Yaskawa INFORM job: A_ROOF_UPPER_0614_2_PAINT_12.JBI

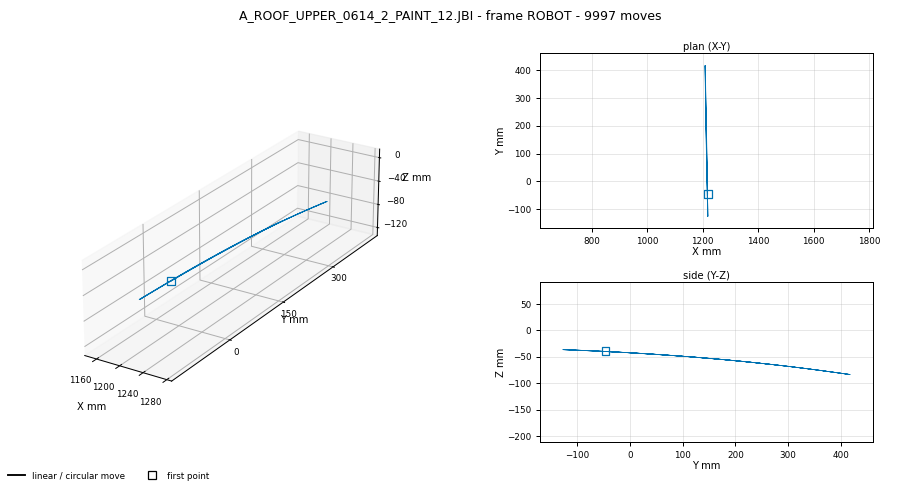
[picture p0: tool path of A_ROOF_UPPER_0614_2_PAINT_12.JBI in frame ROBOT, 9997 of 9997 moves have a stored position in this frame; points joined in program order, loops and branches not executed]
/JOB
//NAME A_ROOF_UPPER_0614_2_PAINT12
//POS
///NPOS 9997,0,0,0,0,0
///TOOL 1
///USER 0
///POSTYPE ROBOT
///RECTAN
///RCONF 1,0,0,0,0,0,0,0,0,0,0,0,0,0,0,0,0,0,0,0,0,0,0,0
C00000=1218.078,-45.969,-39.656,179.952,5.400,148.957
C00001=1218.073,-45.719,-39.668,179.954,5.400,148.956
C00002=1218.068,-45.469,-39.681,179.956,5.401,148.955
C00003=1218.063,-45.220,-39.693,179.959,5.401,148.955
C00004=1218.057,-44.970,-39.705,179.961,5.401,148.954
C00005=1218.052,-44.720,-39.718,179.964,5.401,148.953
C00006=1218.047,-44.471,-39.730,179.966,5.402,148.953
C00007=1218.042,-44.221,-39.742,179.968,5.401,148.952
C00008=1218.037,-43.971,-39.755,179.971,5.402,148.951
C00009=1218.032,-43.722,-39.768,179.973,5.401,148.950
C00010=1218.027,-43.472,-39.780,179.976,5.402,148.950
C00011=1218.022,-43.222,-39.792,179.979,5.402,148.949
C00012=1218.016,-42.973,-39.805,179.981,5.402,148.948
C00013=1218.012,-42.723,-39.818,179.983,5.403,148.948
C00014=1218.007,-42.474,-39.830,179.986,5.403,148.947
C00015=1218.001,-42.224,-39.842,179.988,5.403,148.946
C00016=1217.996,-41.974,-39.856,179.991,5.403,148.945
C00017=1217.990,-41.725,-39.868,179.993,5.404,148.945
C00018=1217.986,-41.475,-39.881,179.995,5.403,148.944
C00019=1217.980,-41.225,-39.893,179.998,5.404,148.943
C00020=1217.975,-40.976,-39.906,-180.000,5.403,148.943
C00021=1217.970,-40.726,-39.918,-179.997,5.404,148.942
C00022=1217.966,-40.476,-39.931,-179.995,5.405,148.942
C00023=1217.961,-40.227,-39.944,-179.993,5.404,148.941
C00024=1217.955,-39.977,-39.956,-179.990,5.405,148.940
C00025=1217.950,-39.728,-39.968,-179.988,5.405,148.939
C00026=1217.944,-39.478,-39.981,-179.985,5.405,148.939
C00027=1217.940,-39.228,-39.994,-179.983,5.406,148.938
C00028=1217.934,-38.979,-40.007,-179.980,5.406,148.937
C00029=1217.929,-38.729,-40.020,-179.978,5.406,148.937
C00030=1217.924,-38.480,-40.032,-179.975,5.406,148.936
C00031=1217.919,-38.229,-40.044,-179.973,5.407,148.935
C00032=1217.914,-37.980,-40.057,-179.971,5.406,148.935
C00033=1217.908,-37.731,-40.070,-179.968,5.407,148.934
C00034=1217.904,-37.481,-40.083,-179.965,5.407,148.933
C00035=1217.899,-37.231,-40.096,-179.963,5.407,148.932
C00036=1217.894,-36.982,-40.108,-179.961,5.407,148.932
C00037=1217.889,-36.733,-40.121,-179.959,5.407,148.931
C00038=1217.883,-36.482,-40.135,-179.956,5.408,148.930
C00039=1217.878,-36.233,-40.147,-179.953,5.408,148.930
C00040=1217.873,-35.984,-40.160,-179.951,5.408,148.929
C00041=1217.868,-35.734,-40.172,-179.948,5.408,148.928
C00042=1217.863,-35.484,-40.185,-179.946,5.409,148.928
C00043=1217.858,-35.235,-40.199,-179.944,5.408,148.927
C00044=1217.852,-34.985,-40.210,-179.941,5.409,148.926
C00045=1217.848,-34.735,-40.223,-179.938,5.409,148.925
C00046=1217.842,-34.485,-40.236,-179.937,5.409,148.925
C00047=1217.837,-34.236,-40.249,-179.934,5.410,148.924
C00048=1217.832,-33.986,-40.262,-179.931,5.410,148.924
C00049=1217.827,-33.736,-40.275,-179.929,5.410,148.923
C00050=1217.822,-33.487,-40.287,-179.927,5.411,148.922
C00051=1217.817,-33.237,-40.301,-179.924,5.411,148.921
C00052=1217.812,-32.988,-40.314,-179.922,5.411,148.921
C00053=1217.807,-32.739,-40.327,-179.919,5.411,148.920
C00054=1217.802,-32.489,-40.340,-179.917,5.412,148.919
C00055=1217.796,-32.239,-40.353,-179.915,5.411,148.919
C00056=1217.791,-31.990,-40.366,-179.912,5.412,148.918
C00057=1217.787,-31.740,-40.379,-179.909,5.412,148.917
C00058=1217.781,-31.490,-40.392,-179.907,5.412,148.917
C00059=1217.776,-31.241,-40.404,-179.904,5.412,148.916
C00060=1217.771,-30.991,-40.417,-179.902,5.413,148.915
C00061=1217.765,-30.741,-40.430,-179.900,5.413,148.914
C00062=1217.760,-30.492,-40.443,-179.897,5.413,148.914
C00063=1217.756,-30.242,-40.456,-179.894,5.414,148.913
C00064=1217.750,-29.992,-40.469,-179.892,5.413,148.912
C00065=1217.745,-29.743,-40.483,-179.890,5.414,148.912
C00066=1217.740,-29.493,-40.496,-179.887,5.414,148.911
C00067=1217.734,-29.244,-40.509,-179.885,5.414,148.910
C00068=1217.730,-28.994,-40.522,-179.882,5.414,148.910
C00069=1217.725,-28.745,-40.534,-179.880,5.415,148.909
C00070=1217.720,-28.494,-40.548,-179.878,5.415,148.908
C00071=1217.715,-28.246,-40.561,-179.875,5.415,148.908
C00072=1217.710,-27.996,-40.574,-179.873,5.416,148.907
C00073=1217.704,-27.746,-40.587,-179.870,5.416,148.906
C00074=1217.699,-27.497,-40.600,-179.868,5.416,148.906
C00075=1217.695,-27.247,-40.613,-179.865,5.417,148.905
C00076=1217.689,-26.998,-40.627,-179.863,5.417,148.904
C00077=1217.684,-26.748,-40.639,-179.861,5.417,148.904
C00078=1217.679,-26.498,-40.653,-179.858,5.417,148.903
C00079=1217.674,-26.249,-40.666,-179.855,5.418,148.902
C00080=1217.669,-25.999,-40.679,-179.853,5.417,148.901
C00081=1217.664,-25.750,-40.692,-179.851,5.418,148.901
C00082=1217.659,-25.499,-40.705,-179.848,5.418,148.900
C00083=1217.653,-25.250,-40.719,-179.846,5.418,148.899
C00084=1217.648,-25.001,-40.732,-179.843,5.419,148.899
C00085=1217.643,-24.751,-40.746,-179.840,5.419,148.898
C00086=1217.638,-24.502,-40.758,-179.838,5.420,148.897
C00087=1217.633,-24.251,-40.772,-179.836,5.419,148.897
C00088=1217.628,-24.002,-40.785,-179.833,5.420,148.896
C00089=1217.623,-23.752,-40.798,-179.830,5.420,148.895
C00090=1217.618,-23.503,-40.811,-179.828,5.420,148.894
C00091=1217.613,-23.253,-40.825,-179.826,5.420,148.894
C00092=1217.607,-22.984,-40.839,-179.823,5.421,148.893
C00093=1217.602,-22.715,-40.854,-179.820,5.421,148.892
C00094=1217.597,-22.445,-40.867,-179.818,5.421,148.892
C00095=1217.591,-22.176,-40.882,-179.816,5.422,148.891
C00096=1217.585,-21.926,-40.896,-179.813,5.422,148.890
C00097=1217.581,-21.677,-40.909,-179.810,5.423,148.890
C00098=1217.575,-21.427,-40.922,-179.808,5.422,148.889
C00099=1217.571,-21.177,-40.935,-179.806,5.423,148.888
C00100=1217.565,-20.928,-40.949,-179.803,5.423,148.888
C00101=1217.561,-20.678,-40.962,-179.800,5.424,148.887
C00102=1217.555,-20.429,-40.976,-179.798,5.423,148.886
C00103=1217.551,-20.179,-40.989,-179.795,5.424,148.885
C00104=1217.545,-19.929,-41.002,-179.793,5.424,148.885
C00105=1217.540,-19.680,-41.016,-179.791,5.424,148.884
C00106=1217.535,-19.430,-41.029,-179.788,5.425,148.883
C00107=1217.530,-19.180,-41.044,-179.785,5.425,148.883
C00108=1217.524,-18.931,-41.056,-179.783,5.426,148.882
C00109=1217.520,-18.681,-41.070,-179.781,5.425,148.881
C00110=1217.514,-18.432,-41.083,-179.778,5.426,148.881
C00111=1217.509,-18.182,-41.097,-179.775,5.426,148.880
C00112=1217.504,-17.933,-41.110,-179.773,5.426,148.879
C00113=1217.499,-17.683,-41.124,-179.771,5.427,148.879
C00114=1217.494,-17.434,-41.137,-179.768,5.427,148.878
C00115=1217.489,-17.184,-41.151,-179.766,5.428,148.877
C00116=1217.484,-16.934,-41.165,-179.764,5.427,148.877
C00117=1217.479,-16.685,-41.178,-179.761,5.428,148.876
C00118=1217.474,-16.435,-41.192,-179.758,5.428,148.875
C00119=1217.468,-16.186,-41.205,-179.756,5.428,148.875
C00120=1217.464,-15.936,-41.218,-179.754,5.429,148.874
C00121=1217.458,-15.687,-41.232,-179.751,5.429,148.873
C00122=1217.453,-15.437,-41.246,-179.748,5.430,148.872
C00123=1217.449,-15.187,-41.260,-179.746,5.429,148.872
C00124=1217.443,-14.938,-41.273,-179.744,5.430,148.871
C00125=1217.438,-14.688,-41.287,-179.741,5.430,148.870
C00126=1217.433,-14.439,-41.300,-179.738,5.431,148.870
C00127=1217.428,-14.189,-41.314,-179.736,5.431,148.869
C00128=1217.423,-13.939,-41.328,-179.734,5.431,148.868
C00129=1217.418,-13.690,-41.341,-179.731,5.432,148.868
C00130=1217.413,-13.440,-41.355,-179.729,5.431,148.867
C00131=1217.407,-13.191,-41.369,-179.726,5.432,148.866
C00132=1217.403,-12.941,-41.382,-179.724,5.432,148.866
C00133=1217.398,-12.691,-41.396,-179.721,5.433,148.865
C00134=1217.392,-12.442,-41.410,-179.719,5.433,148.864
C00135=1217.387,-12.192,-41.424,-179.717,5.433,148.864
C00136=1217.383,-11.943,-41.437,-179.714,5.434,148.863
C00137=1217.377,-11.694,-41.451,-179.711,5.434,148.862
C00138=1217.372,-11.443,-41.465,-179.709,5.434,148.862
C00139=1217.368,-11.194,-41.479,-179.707,5.434,148.861
C00140=1217.362,-10.945,-41.492,-179.704,5.435,148.860
C00141=1217.357,-10.695,-41.507,-179.701,5.435,148.860
C00142=1217.351,-10.446,-41.520,-179.699,5.435,148.859
C00143=1217.347,-10.196,-41.534,-179.697,5.436,148.858
C00144=1217.342,-9.946,-41.548,-179.694,5.436,148.857
C00145=1217.336,-9.697,-41.561,-179.691,5.437,148.857
C00146=1217.331,-9.447,-41.575,-179.689,5.436,148.856
C00147=1217.327,-9.198,-41.589,-179.686,5.437,148.855
C00148=1217.322,-8.948,-41.603,-179.684,5.437,148.855
C00149=1217.317,-8.699,-41.617,-179.681,5.438,148.854
C00150=1217.311,-8.449,-41.631,-179.679,5.438,148.853
C00151=1217.307,-8.199,-41.645,-179.676,5.438,148.853
C00152=1217.302,-7.950,-41.658,-179.674,5.439,148.852
C00153=1217.297,-7.701,-41.673,-179.672,5.439,148.851
C00154=1217.291,-7.450,-41.686,-179.670,5.439,148.851
C00155=1217.286,-7.201,-41.700,-179.667,5.440,148.850
C00156=1217.281,-6.951,-41.714,-179.664,5.440,148.849
C00157=1217.276,-6.702,-41.729,-179.662,5.441,148.849
C00158=1217.272,-6.452,-41.742,-179.660,5.440,148.848
C00159=1217.266,-6.203,-41.756,-179.657,5.441,148.847
C00160=1217.261,-5.954,-41.771,-179.654,5.441,148.847
C00161=1217.256,-5.703,-41.784,-179.652,5.442,148.846
C00162=1217.250,-5.454,-41.798,-179.649,5.442,148.845
C00163=1217.246,-5.205,-41.812,-179.647,5.442,148.845
C00164=1217.241,-4.955,-41.827,-179.644,5.443,148.844
C00165=1217.236,-4.705,-41.840,-179.641,5.443,148.843
C00166=1217.231,-4.456,-41.854,-179.639,5.444,148.842
C00167=1217.226,-4.207,-41.868,-179.637,5.443,148.842
C00168=1217.221,-3.957,-41.883,-179.634,5.444,148.841
C00169=1217.216,-3.707,-41.897,-179.632,5.445,148.841
C00170=1217.210,-3.458,-41.911,-179.629,5.445,148.840
C00171=1217.205,-3.208,-41.924,-179.627,5.445,148.839
C00172=1217.200,-2.958,-41.939,-179.625,5.445,148.839
C00173=1217.195,-2.709,-41.953,-179.622,5.446,148.838
C00174=1217.190,-2.460,-41.967,-179.619,5.446,148.837
C00175=1217.185,-2.210,-41.981,-179.617,5.446,148.837
C00176=1217.180,-1.960,-41.995,-179.615,5.447,148.836
C00177=1217.176,-1.711,-42.009,-179.612,5.447,148.835
C00178=1217.171,-1.461,-42.023,-179.609,5.448,148.834
C00179=1217.165,-1.212,-42.037,-179.607,5.448,148.834
C00180=1217.160,-0.962,-42.052,-179.604,5.448,148.833
C00181=1217.155,-0.713,-42.066,-179.602,5.448,148.832
C00182=1217.150,-0.463,-42.080,-179.599,5.449,148.832
C00183=1217.145,-0.213,-42.094,-179.597,5.449,148.831
C00184=1217.140,0.036,-42.108,-179.594,5.450,148.830
C00185=1217.135,0.286,-42.123,-179.592,5.450,148.830
C00186=1217.130,0.535,-42.138,-179.590,5.450,148.829
C00187=1217.125,0.784,-42.152,-179.587,5.451,148.828
C00188=1217.120,1.034,-42.166,-179.584,5.452,148.828
C00189=1217.115,1.283,-42.180,-179.582,5.451,148.827
C00190=1217.110,1.533,-42.194,-179.580,5.452,148.826
C00191=1217.105,1.782,-42.209,-179.577,5.452,148.826
C00192=1217.100,2.032,-42.223,-179.574,5.453,148.825
C00193=1217.095,2.282,-42.237,-179.572,5.453,148.824
C00194=1217.090,2.532,-42.251,-179.570,5.453,148.824
C00195=1217.084,2.781,-42.265,-179.567,5.453,148.823
C00196=1217.078,3.050,-42.282,-179.564,5.454,148.822
C00197=1217.073,3.319,-42.297,-179.562,5.455,148.822
C00198=1217.068,3.588,-42.312,-179.559,5.455,148.821
C00199=1217.063,3.857,-42.328,-179.556,5.456,148.820
C00200=1217.058,4.106,-42.342,-179.554,5.456,148.820
C00201=1217.053,4.356,-42.357,-179.551,5.457,148.819
C00202=1217.048,4.606,-42.371,-179.549,5.456,148.818
C00203=1217.043,4.854,-42.386,-179.546,5.457,148.817
C00204=1217.038,5.104,-42.400,-179.544,5.457,148.817
C00205=1217.032,5.354,-42.415,-179.541,5.458,148.816
C00206=1217.027,5.604,-42.429,-179.538,5.458,148.815
C00207=1217.022,5.853,-42.444,-179.536,5.458,148.815
C00208=1217.017,6.102,-42.458,-179.534,5.459,148.814
C00209=1217.012,6.352,-42.473,-179.531,5.459,148.813
C00210=1217.007,6.602,-42.487,-179.528,5.460,148.813
C00211=1217.002,6.852,-42.501,-179.526,5.460,148.812
C00212=1216.997,7.100,-42.516,-179.524,5.460,148.812
C00213=1216.992,7.350,-42.531,-179.521,5.461,148.811
C00214=1216.987,7.600,-42.545,-179.519,5.461,148.810
C00215=1216.982,7.849,-42.560,-179.516,5.462,148.809
C00216=1216.977,8.099,-42.574,-179.513,5.462,148.809
C00217=1216.972,8.348,-42.588,-179.511,5.463,148.808
C00218=1216.967,8.597,-42.603,-179.509,5.462,148.807
C00219=1216.962,8.847,-42.618,-179.506,5.463,148.807
C00220=1216.957,9.097,-42.633,-179.503,5.464,148.806
C00221=1216.952,9.346,-42.648,-179.501,5.464,148.805
C00222=1216.947,9.596,-42.662,-179.498,5.465,148.805
C00223=1216.942,9.846,-42.676,-179.496,5.464,148.804
C00224=1216.937,10.095,-42.692,-179.494,5.465,148.804
C00225=1216.932,10.345,-42.706,-179.491,5.466,148.803
C00226=1216.927,10.594,-42.720,-179.489,5.466,148.802
C00227=1216.922,10.843,-42.735,-179.486,5.467,148.801
C00228=1216.917,11.093,-42.750,-179.483,5.467,148.801
C00229=1216.912,11.343,-42.765,-179.481,5.467,148.800
C00230=1216.907,11.592,-42.779,-179.479,5.467,148.799
C00231=1216.901,11.841,-42.793,-179.476,5.468,148.799
C00232=1216.897,12.090,-42.808,-179.473,5.469,148.798
C00233=1216.891,12.340,-42.823,-179.471,5.469,148.797
C00234=1216.886,12.590,-42.838,-179.468,5.470,148.797
C00235=1216.881,12.839,-42.852,-179.466,5.469,148.796
C00236=1216.876,13.089,-42.868,-179.464,5.470,148.796
C00237=1216.871,13.338,-42.882,-179.461,5.471,148.795
C00238=1216.866,13.588,-42.897,-179.458,5.471,148.794
C00239=1216.861,13.837,-42.912,-179.456,5.472,148.793
C00240=1216.856,14.087,-42.926,-179.453,5.472,148.793
C00241=1216.851,14.336,-42.941,-179.450,5.473,148.792
C00242=1216.847,14.587,-42.956,-179.448,5.472,148.791
C00243=1216.841,14.836,-42.972,-179.446,5.473,148.791
C00244=1216.836,15.086,-42.986,-179.443,5.474,148.790
C00245=1216.832,15.335,-43.001,-179.440,5.474,148.789
C00246=1216.826,15.584,-43.017,-179.438,5.475,148.789
C00247=1216.821,15.834,-43.031,-179.436,5.475,148.788
C00248=1216.817,16.083,-43.046,-179.434,5.475,148.788
C00249=1216.811,16.333,-43.061,-179.431,5.476,148.787
C00250=1216.806,16.582,-43.076,-179.428,5.476,148.786
C00251=1216.802,16.832,-43.090,-179.426,5.477,148.785
C00252=1216.796,17.081,-43.106,-179.423,5.477,148.785
C00253=1216.791,17.330,-43.121,-179.420,5.478,148.784
C00254=1216.787,17.580,-43.135,-179.418,5.478,148.783
C00255=1216.781,17.830,-43.150,-179.416,5.478,148.783
C00256=1216.776,18.079,-43.165,-179.413,5.479,148.782
C00257=1216.771,18.329,-43.180,-179.411,5.479,148.782
C00258=1216.766,18.578,-43.195,-179.408,5.480,148.781
C00259=1216.761,18.827,-43.210,-179.406,5.481,148.780
C00260=1216.756,19.078,-43.225,-179.403,5.481,148.780
C00261=1216.752,19.327,-43.240,-179.400,5.482,148.779
C00262=1216.746,19.577,-43.255,-179.398,5.481,148.778
C00263=1216.741,19.826,-43.270,-179.396,5.482,148.778
C00264=1216.736,20.075,-43.286,-179.393,5.482,148.777
C00265=1216.731,20.325,-43.300,-179.390,5.483,148.776
C00266=1216.726,20.574,-43.315,-179.388,5.483,148.775
C00267=1216.721,20.823,-43.331,-179.385,5.484,148.775
C00268=1216.716,21.073,-43.345,-179.383,5.485,148.774
C00269=1216.711,21.322,-43.361,-179.380,5.485,148.774
C00270=1216.707,21.572,-43.376,-179.378,5.485,148.773
C00271=1216.701,21.822,-43.392,-179.375,5.486,148.772
C00272=1216.696,22.071,-43.406,-179.373,5.486,148.772
C00273=1216.691,22.321,-43.421,-179.370,5.487,148.771
C00274=1216.686,22.570,-43.436,-179.367,5.487,148.770
C00275=1216.681,22.819,-43.452,-179.365,5.488,148.770
C00276=1216.676,23.069,-43.466,-179.363,5.489,148.769
C00277=1216.671,23.319,-43.482,-179.360,5.489,148.768
C00278=1216.666,23.568,-43.497,-179.357,5.490,148.768
C00279=1216.661,23.818,-43.513,-179.355,5.489,148.767
C00280=1216.656,24.067,-43.528,-179.353,5.490,148.766
C00281=1216.651,24.317,-43.543,-179.350,5.490,148.766
C00282=1216.646,24.566,-43.558,-179.347,5.491,148.765
C00283=1216.641,24.816,-43.574,-179.345,5.492,148.764
C00284=1216.637,25.065,-43.589,-179.342,5.492,148.764
C00285=1216.631,25.314,-43.604,-179.340,5.493,148.763
C00286=1216.626,25.564,-43.620,-179.337,5.494,148.763
C00287=1216.621,25.813,-43.635,-179.335,5.494,148.762
C00288=1216.616,26.064,-43.650,-179.333,5.494,148.761
C00289=1216.612,26.313,-43.665,-179.330,5.494,148.761
C00290=1216.606,26.562,-43.681,-179.327,5.495,148.760
C00291=1216.601,26.811,-43.696,-179.325,5.495,148.759
C00292=1216.596,27.061,-43.711,-179.322,5.496,148.758
C00293=1216.591,27.311,-43.727,-179.319,5.496,148.758
C00294=1216.587,27.560,-43.742,-179.317,5.497,148.757
C00295=1216.581,27.809,-43.758,-179.315,5.498,148.757
C00296=1216.576,28.059,-43.773,-179.312,5.498,148.756
C00297=1216.571,28.308,-43.788,-179.309,5.499,148.755
C00298=1216.566,28.558,-43.804,-179.307,5.499,148.755
C00299=1216.562,28.807,-43.819,-179.305,5.499,148.754
C00300=1216.556,29.076,-43.836,-179.302,5.500,148.753
C00301=1216.550,29.344,-43.853,-179.299,5.500,148.753
C00302=1216.545,29.613,-43.870,-179.297,5.501,148.752
C00303=1216.540,29.882,-43.885,-179.293,5.502,148.751
C00304=1216.535,30.132,-43.901,-179.291,5.502,148.751
C00305=1216.530,30.381,-43.917,-179.289,5.502,148.750
C00306=1216.525,30.630,-43.932,-179.286,5.503,148.749
C00307=1216.519,30.880,-43.947,-179.283,5.503,148.749
C00308=1216.515,31.130,-43.963,-179.281,5.504,148.748
C00309=1216.510,31.378,-43.979,-179.279,5.505,148.747
C00310=1216.505,31.628,-43.995,-179.276,5.505,148.747
C00311=1216.500,31.877,-44.010,-179.273,5.506,148.746
C00312=1216.496,32.127,-44.026,-179.271,5.507,148.745
C00313=1216.490,32.376,-44.041,-179.268,5.507,148.745
C00314=1216.485,32.626,-44.057,-179.265,5.508,148.744
C00315=1216.480,32.876,-44.073,-179.263,5.508,148.743
C00316=1216.475,33.125,-44.088,-179.261,5.508,148.743
C00317=1216.470,33.374,-44.103,-179.259,5.509,148.742
C00318=1216.465,33.624,-44.119,-179.256,5.509,148.742
C00319=1216.460,33.873,-44.136,-179.253,5.510,148.741
C00320=1216.455,34.122,-44.151,-179.251,5.510,148.740
C00321=1216.450,34.372,-44.166,-179.248,5.511,148.740
C00322=1216.445,34.622,-44.182,-179.245,5.511,148.739
C00323=1216.440,34.871,-44.198,-179.243,5.512,148.738
C00324=1216.435,35.120,-44.213,-179.241,5.513,148.738
C00325=1216.431,35.370,-44.229,-179.238,5.513,148.737
C00326=1216.425,35.619,-44.245,-179.235,5.514,148.736
C00327=1216.420,35.869,-44.261,-179.233,5.515,148.736
C00328=1216.415,36.119,-44.277,-179.230,5.515,148.735
C00329=1216.411,36.368,-44.292,-179.227,5.516,148.734
C00330=1216.406,36.617,-44.308,-179.225,5.517,148.734
C00331=1216.401,36.867,-44.324,-179.223,5.517,148.733
C00332=1216.395,37.116,-44.339,-179.220,5.517,148.733
C00333=1216.390,37.366,-44.355,-179.218,5.517,148.732
C00334=1216.385,37.615,-44.372,-179.215,5.518,148.731
C00335=1216.381,37.864,-44.387,-179.213,5.518,148.731
C00336=1216.376,38.114,-44.403,-179.210,5.519,148.730
C00337=1216.371,38.364,-44.418,-179.208,5.520,148.729
C00338=1216.366,38.612,-44.434,-179.205,5.520,148.729
C00339=1216.361,38.862,-44.450,-179.202,5.521,148.728
C00340=1216.355,39.112,-44.466,-179.200,5.522,148.727
C00341=1216.351,39.361,-44.483,-179.197,5.522,148.727
C00342=1216.345,39.611,-44.498,-179.195,5.523,148.726
C00343=1216.341,39.860,-44.513,-179.192,5.523,148.725
C00344=1216.336,40.109,-44.530,-179.190,5.524,148.725
C00345=1216.331,40.359,-44.545,-179.187,5.525,148.724
C00346=1216.326,40.609,-44.561,-179.184,5.525,148.724
C00347=1216.321,40.858,-44.578,-179.182,5.526,148.723
C00348=1216.316,41.107,-44.593,-179.179,5.526,148.722
C00349=1216.311,41.357,-44.609,-179.177,5.527,148.722
C00350=1216.306,41.606,-44.626,-179.174,5.528,148.721
C00351=1216.301,41.856,-44.642,-179.172,5.528,148.720
C00352=1216.296,42.105,-44.658,-179.169,5.529,148.720
C00353=1216.291,42.355,-44.674,-179.166,5.529,148.719
C00354=1216.286,42.604,-44.689,-179.164,5.530,148.718
C00355=1216.281,42.853,-44.706,-179.161,5.530,148.718
C00356=1216.276,43.103,-44.722,-179.159,5.531,148.717
C00357=1216.271,43.352,-44.738,-179.157,5.531,148.717
C00358=1216.266,43.602,-44.754,-179.154,5.532,148.716
C00359=1216.261,43.851,-44.770,-179.152,5.532,148.715
C00360=1216.256,44.101,-44.786,-179.149,5.533,148.715
C00361=1216.251,44.350,-44.802,-179.146,5.533,148.714
C00362=1216.246,44.600,-44.818,-179.144,5.534,148.713
C00363=1216.241,44.849,-44.835,-179.142,5.535,148.713
C00364=1216.236,45.099,-44.851,-179.139,5.535,148.712
C00365=1216.231,45.347,-44.867,-179.136,5.536,148.711
C00366=1216.227,45.598,-44.883,-179.134,5.536,148.711
C00367=1216.222,45.846,-44.899,-179.131,5.537,148.710
C00368=1216.217,46.096,-44.915,-179.129,5.538,148.710
C00369=1216.212,46.345,-44.931,-179.126,5.538,148.709
C00370=1216.207,46.595,-44.947,-179.124,5.539,148.708
C00371=1216.202,46.844,-44.964,-179.121,5.540,148.708
C00372=1216.197,47.094,-44.980,-179.118,5.540,148.707
C00373=1216.192,47.343,-44.996,-179.116,5.541,148.707
C00374=1216.187,47.592,-45.013,-179.114,5.542,148.706
C00375=1216.182,47.842,-45.028,-179.111,5.542,148.705
C00376=1216.178,48.091,-45.045,-179.108,5.543,148.705
C00377=1216.172,48.340,-45.061,-179.106,5.543,148.704
C00378=1216.168,48.590,-45.077,-179.103,5.544,148.703
C00379=1216.162,48.839,-45.094,-179.101,5.545,148.703
C00380=1216.157,49.089,-45.111,-179.098,5.545,148.702
C00381=1216.152,49.338,-45.126,-179.096,5.546,148.701
C00382=1216.148,49.588,-45.143,-179.093,5.546,148.701
C00383=1216.143,49.838,-45.159,-179.090,5.547,148.700
C00384=1216.138,50.087,-45.175,-179.088,5.548,148.700
C00385=1216.133,50.336,-45.192,-179.086,5.548,148.699
C00386=1216.128,50.585,-45.208,-179.083,5.549,148.698
C00387=1216.123,50.835,-45.225,-179.080,5.549,148.698
C00388=1216.118,51.084,-45.241,-179.078,5.550,148.697
C00389=1216.113,51.334,-45.258,-179.075,5.551,148.696
C00390=1216.108,51.584,-45.274,-179.073,5.551,148.696
C00391=1216.103,51.832,-45.290,-179.070,5.552,148.695
C00392=1216.099,52.082,-45.307,-179.068,5.553,148.695
C00393=1216.093,52.331,-45.324,-179.065,5.553,148.694
C00394=1216.088,52.581,-45.340,-179.062,5.554,148.693
C00395=1216.084,52.831,-45.356,-179.060,5.555,148.693
C00396=1216.079,53.079,-45.373,-179.058,5.555,148.692
C00397=1216.074,53.329,-45.389,-179.055,5.556,148.691
C00398=1216.068,53.578,-45.406,-179.052,5.556,148.691
C00399=1216.063,53.828,-45.422,-179.050,5.557,148.690
C00400=1216.059,54.078,-45.439,-179.047,5.559,148.690
C00401=1216.054,54.326,-45.455,-179.044,5.559,148.689
C00402=1216.049,54.576,-45.472,-179.042,5.560,148.688
C00403=1216.044,54.826,-45.489,-179.039,5.560,148.688
C00404=1216.039,55.094,-45.506,-179.036,5.561,148.687
C00405=1216.033,55.362,-45.524,-179.034,5.561,148.686
C00406=1216.028,55.631,-45.542,-179.031,5.562,148.686
C00407=1216.022,55.899,-45.559,-179.028,5.562,148.685
C00408=1216.018,56.149,-45.576,-179.026,5.563,148.684
C00409=1216.013,56.399,-45.593,-179.024,5.564,148.684
C00410=1216.008,56.647,-45.610,-179.021,5.564,148.683
C00411=1216.003,56.897,-45.626,-179.018,5.566,148.683
C00412=1215.998,57.147,-45.644,-179.015,5.566,148.682
C00413=1215.993,57.395,-45.660,-179.013,5.567,148.681
C00414=1215.988,57.645,-45.677,-179.010,5.568,148.681
C00415=1215.983,57.895,-45.694,-179.008,5.568,148.680
C00416=1215.978,58.143,-45.710,-179.005,5.569,148.679
C00417=1215.974,58.393,-45.727,-179.003,5.570,148.679
C00418=1215.968,58.643,-45.744,-179.000,5.571,148.678
C00419=1215.963,58.892,-45.760,-178.998,5.571,148.678
C00420=1215.959,59.141,-45.777,-178.995,5.572,148.677
C00421=1215.954,59.391,-45.794,-178.992,5.572,148.676
C00422=1215.949,59.640,-45.811,-178.990,5.573,148.676
C00423=1215.944,59.889,-45.827,-178.988,5.574,148.675
C00424=1215.939,60.139,-45.845,-178.985,5.574,148.675
C00425=1215.934,60.388,-45.861,-178.982,5.575,148.674
C00426=1215.929,60.637,-45.878,-178.980,5.575,148.673
C00427=1215.924,60.887,-45.895,-178.978,5.576,148.673
C00428=1215.920,61.136,-45.911,-178.975,5.577,148.672
C00429=1215.914,61.386,-45.929,-178.972,5.577,148.671
C00430=1215.909,61.635,-45.945,-178.969,5.579,148.671
C00431=1215.904,61.885,-45.962,-178.967,5.579,148.670
C00432=1215.900,62.134,-45.979,-178.964,5.580,148.670
C00433=1215.895,62.384,-45.996,-178.962,5.581,148.669
C00434=1215.889,62.633,-46.013,-178.959,5.581,148.668
C00435=1215.885,62.882,-46.030,-178.957,5.582,148.668
C00436=1215.880,63.132,-46.047,-178.954,5.583,148.667
C00437=1215.875,63.381,-46.064,-178.952,5.583,148.667
C00438=1215.870,63.630,-46.081,-178.949,5.584,148.666
C00439=1215.865,63.880,-46.097,-178.946,5.585,148.665
C00440=1215.860,64.129,-46.115,-178.944,5.586,148.665
C00441=1215.855,64.379,-46.131,-178.942,5.586,148.664
C00442=1215.850,64.627,-46.149,-178.939,5.587,148.664
C00443=1215.845,64.877,-46.166,-178.936,5.587,148.663
C00444=1215.840,65.127,-46.183,-178.934,5.589,148.662
C00445=1215.836,65.376,-46.200,-178.931,5.590,148.662
C00446=1215.830,65.626,-46.217,-178.928,5.590,148.661
C00447=1215.826,65.874,-46.234,-178.926,5.591,148.660
C00448=1215.820,66.124,-46.251,-178.924,5.592,148.660
C00449=1215.816,66.373,-46.268,-178.921,5.592,148.659
C00450=1215.811,66.623,-46.285,-178.918,5.593,148.659
C00451=1215.807,66.872,-46.302,-178.916,5.593,148.658
C00452=1215.801,67.122,-46.320,-178.914,5.594,148.658
C00453=1215.796,67.371,-46.336,-178.911,5.595,148.657
C00454=1215.791,67.620,-46.353,-178.908,5.595,148.656
C00455=1215.787,67.869,-46.371,-178.905,5.597,148.656
C00456=1215.782,68.119,-46.388,-178.903,5.598,148.655
C00457=1215.777,68.369,-46.405,-178.900,5.598,148.655
C00458=1215.772,68.618,-46.423,-178.898,5.599,148.654
C00459=1215.767,68.867,-46.439,-178.895,5.599,148.653
C00460=1215.762,69.116,-46.456,-178.893,5.600,148.653
C00461=1215.757,69.365,-46.474,-178.890,5.601,148.652
C00462=1215.753,69.615,-46.491,-178.888,5.601,148.651
C00463=1215.747,69.865,-46.508,-178.885,5.602,148.651
C00464=1215.743,70.114,-46.526,-178.883,5.603,148.650
C00465=1215.738,70.363,-46.543,-178.880,5.604,148.650
C00466=1215.733,70.613,-46.561,-178.877,5.605,148.649
C00467=1215.728,70.861,-46.577,-178.875,5.605,148.648
C00468=1215.723,71.111,-46.594,-178.872,5.606,148.648
C00469=1215.718,71.360,-46.612,-178.870,5.607,148.647
C00470=1215.713,71.610,-46.629,-178.867,5.608,148.647
C00471=1215.709,71.859,-46.647,-178.865,5.608,148.646
C00472=1215.703,72.109,-46.664,-178.862,5.609,148.646
C00473=1215.699,72.358,-46.681,-178.860,5.610,148.645
C00474=1215.694,72.607,-46.699,-178.857,5.611,148.644
C00475=1215.689,72.857,-46.716,-178.854,5.612,148.644
C00476=1215.684,73.106,-46.734,-178.852,5.612,148.643
C00477=1215.679,73.355,-46.750,-178.849,5.613,148.642
C00478=1215.674,73.604,-46.768,-178.847,5.614,148.642
C00479=1215.669,73.854,-46.786,-178.844,5.615,148.641
C00480=1215.664,74.103,-46.803,-178.842,5.615,148.641
C00481=1215.659,74.353,-46.820,-178.839,5.616,148.640
C00482=1215.654,74.602,-46.838,-178.836,5.617,148.640
C00483=1215.649,74.851,-46.856,-178.834,5.618,148.639
C00484=1215.645,75.101,-46.873,-178.831,5.619,148.638
C00485=1215.640,75.350,-46.891,-178.829,5.619,148.638
C00486=1215.635,75.600,-46.908,-178.826,5.620,148.637
C00487=1215.631,75.849,-46.925,-178.824,5.621,148.637
C00488=1215.625,76.098,-46.943,-178.821,5.621,148.636
C00489=1215.620,76.347,-46.961,-178.818,5.623,148.636
C00490=1215.616,76.597,-46.979,-178.816,5.624,148.635
C00491=1215.610,76.846,-46.996,-178.813,5.624,148.634
C00492=1215.606,77.095,-47.013,-178.811,5.625,148.634
C00493=1215.601,77.345,-47.031,-178.808,5.626,148.633
C00494=1215.596,77.594,-47.049,-178.806,5.626,148.632
C00495=1215.591,77.843,-47.067,-178.803,5.627,148.632
C00496=1215.586,78.093,-47.084,-178.800,5.629,148.631
C00497=1215.582,78.342,-47.101,-178.798,5.629,148.631
C00498=1215.577,78.591,-47.119,-178.795,5.630,148.630
C00499=1215.572,78.841,-47.136,-178.793,5.630,148.629
C00500=1215.567,79.090,-47.154,-178.790,5.631,148.629
C00501=1215.562,79.339,-47.172,-178.788,5.632,148.628
C00502=1215.557,79.589,-47.190,-178.785,5.633,148.628
C00503=1215.552,79.838,-47.207,-178.783,5.634,148.627
C00504=1215.547,80.087,-47.225,-178.780,5.635,148.627
C00505=1215.543,80.336,-47.243,-178.777,5.635,148.626
C00506=1215.537,80.586,-47.260,-178.775,5.636,148.626
C00507=1215.532,80.835,-47.278,-178.772,5.637,148.625
C00508=1215.527,81.104,-47.298,-178.769,5.638,148.624
C00509=1215.522,81.373,-47.316,-178.767,5.639,148.624
C00510=1215.517,81.641,-47.336,-178.764,5.639,148.623
C00511=1215.512,81.909,-47.355,-178.761,5.641,148.622
C00512=1215.507,82.158,-47.373,-178.759,5.642,148.622
C00513=1215.502,82.408,-47.390,-178.756,5.642,148.621
C00514=1215.497,82.657,-47.408,-178.753,5.643,148.621
C00515=1215.492,82.906,-47.426,-178.751,5.644,148.620
C00516=1215.487,83.156,-47.444,-178.748,5.645,148.619
C00517=1215.482,83.405,-47.462,-178.746,5.646,148.619
C00518=1215.477,83.654,-47.480,-178.743,5.647,148.618
C00519=1215.473,83.903,-47.497,-178.741,5.647,148.618
C00520=1215.468,84.153,-47.515,-178.738,5.648,148.617
C00521=1215.463,84.402,-47.533,-178.736,5.648,148.616
C00522=1215.458,84.651,-47.551,-178.733,5.650,148.616
C00523=1215.454,84.901,-47.569,-178.730,5.651,148.615
C00524=1215.449,85.150,-47.587,-178.728,5.651,148.615
C00525=1215.444,85.399,-47.605,-178.725,5.652,148.614
C00526=1215.439,85.648,-47.623,-178.723,5.653,148.614
C00527=1215.434,85.897,-47.641,-178.720,5.654,148.613
C00528=1215.429,86.147,-47.659,-178.717,5.655,148.613
C00529=1215.424,86.396,-47.677,-178.715,5.656,148.612
C00530=1215.419,86.645,-47.695,-178.712,5.656,148.611
C00531=1215.415,86.895,-47.713,-178.710,5.657,148.611
C00532=1215.410,87.144,-47.731,-178.707,5.659,148.610
C00533=1215.405,87.394,-47.749,-178.704,5.659,148.609
C00534=1215.399,87.643,-47.767,-178.702,5.660,148.609
C00535=1215.394,87.893,-47.785,-178.700,5.661,148.608
C00536=1215.390,88.141,-47.804,-178.697,5.661,148.608
C00537=1215.385,88.391,-47.822,-178.694,5.663,148.607
C00538=1215.380,88.640,-47.840,-178.692,5.664,148.607
C00539=1215.375,88.889,-47.858,-178.689,5.664,148.606
C00540=1215.370,89.138,-47.876,-178.687,5.665,148.606
C00541=1215.366,89.388,-47.894,-178.684,5.666,148.605
C00542=1215.361,89.637,-47.912,-178.682,5.668,148.605
C00543=1215.356,89.887,-47.931,-178.679,5.668,148.604
C00544=1215.351,90.136,-47.949,-178.676,5.669,148.603
C00545=1215.346,90.385,-47.967,-178.674,5.670,148.603
C00546=1215.341,90.635,-47.985,-178.672,5.670,148.602
C00547=1215.336,90.884,-48.003,-178.668,5.672,148.602
C00548=1215.332,91.134,-48.021,-178.666,5.673,148.601
C00549=1215.327,91.382,-48.040,-178.664,5.673,148.600
C00550=1215.322,91.631,-48.058,-178.661,5.674,148.600
C00551=1215.317,91.881,-48.076,-178.658,5.676,148.599
C00552=1215.312,92.130,-48.095,-178.656,5.676,148.599
C00553=1215.307,92.380,-48.113,-178.653,5.677,148.598
C00554=1215.302,92.629,-48.131,-178.651,5.678,148.598
C00555=1215.298,92.878,-48.150,-178.648,5.678,148.597
C00556=1215.293,93.127,-48.168,-178.645,5.680,148.596
C00557=1215.289,93.377,-48.186,-178.643,5.681,148.596
C00558=1215.283,93.626,-48.205,-178.640,5.681,148.595
C00559=1215.278,93.875,-48.223,-178.638,5.682,148.595
C00560=1215.273,94.124,-48.241,-178.635,5.684,148.594
C00561=1215.269,94.374,-48.260,-178.632,5.684,148.594
C00562=1215.264,94.623,-48.278,-178.630,5.685,148.593
C00563=1215.258,94.872,-48.296,-178.628,5.686,148.593
C00564=1215.254,95.121,-48.315,-178.624,5.687,148.592
C00565=1215.250,95.371,-48.333,-178.622,5.688,148.591
C00566=1215.245,95.620,-48.351,-178.620,5.689,148.591
C00567=1215.239,95.870,-48.370,-178.618,5.690,148.590
C00568=1215.235,96.119,-48.389,-178.614,5.691,148.590
C00569=1215.230,96.368,-48.407,-178.612,5.692,148.589
C00570=1215.224,96.617,-48.425,-178.610,5.693,148.589
C00571=1215.220,96.866,-48.444,-178.607,5.693,148.588
C00572=1215.216,97.116,-48.462,-178.604,5.695,148.587
C00573=1215.211,97.365,-48.480,-178.602,5.696,148.587
C00574=1215.205,97.614,-48.500,-178.599,5.696,148.586
C00575=1215.201,97.864,-48.518,-178.597,5.697,148.586
C00576=1215.196,98.112,-48.537,-178.594,5.699,148.585
C00577=1215.191,98.362,-48.555,-178.591,5.699,148.585
C00578=1215.186,98.612,-48.574,-178.589,5.700,148.584
C00579=1215.182,98.860,-48.592,-178.586,5.701,148.584
C00580=1215.176,99.110,-48.611,-178.584,5.702,148.583
C00581=1215.172,99.359,-48.630,-178.581,5.703,148.583
C00582=1215.167,99.608,-48.648,-178.578,5.704,148.582
C00583=1215.162,99.858,-48.667,-178.576,5.705,148.581
C00584=1215.158,100.107,-48.686,-178.573,5.706,148.581
C00585=1215.153,100.356,-48.704,-178.571,5.707,148.580
C00586=1215.147,100.605,-48.723,-178.568,5.708,148.580
C00587=1215.143,100.855,-48.741,-178.565,5.709,148.579
C00588=1215.138,101.104,-48.760,-178.563,5.710,148.579
C00589=1215.133,101.354,-48.779,-178.560,5.710,148.578
C00590=1215.129,101.602,-48.798,-178.558,5.711,148.578
C00591=1215.123,101.852,-48.816,-178.555,5.713,148.577
C00592=1215.119,102.101,-48.835,-178.553,5.713,148.576
C00593=1215.113,102.350,-48.854,-178.550,5.714,148.576
C00594=1215.109,102.599,-48.872,-178.547,5.716,148.575
C00595=1215.104,102.849,-48.891,-178.545,5.717,148.575
C00596=1215.099,103.098,-48.910,-178.542,5.717,148.574
C00597=1215.095,103.347,-48.929,-178.540,5.718,148.574
C00598=1215.090,103.596,-48.948,-178.537,5.720,148.573
C00599=1215.085,103.845,-48.966,-178.535,5.720,148.573
C00600=1215.080,104.095,-48.985,-178.532,5.721,148.572
C00601=1215.075,104.344,-49.004,-178.529,5.723,148.572
C00602=1215.071,104.593,-49.024,-178.527,5.724,148.571
C00603=1215.066,104.842,-49.042,-178.525,5.724,148.570
C00604=1215.061,105.092,-49.061,-178.522,5.725,148.570
C00605=1215.056,105.341,-49.080,-178.519,5.727,148.569
C00606=1215.051,105.590,-49.099,-178.517,5.727,148.569
C00607=1215.047,105.839,-49.118,-178.514,5.728,148.568
C00608=1215.041,106.088,-49.137,-178.511,5.730,148.568
C00609=1215.037,106.338,-49.155,-178.509,5.730,148.567
C00610=1215.032,106.587,-49.175,-178.507,5.731,148.567
C00611=1215.028,106.836,-49.194,-178.503,5.733,148.566
C00612=1215.022,107.105,-49.214,-178.501,5.734,148.566
C00613=1215.017,107.373,-49.235,-178.498,5.735,148.565
C00614=1215.011,107.642,-49.255,-178.495,5.736,148.564
C00615=1215.007,107.910,-49.275,-178.492,5.737,148.564
C00616=1215.002,108.159,-49.295,-178.490,5.738,148.563
C00617=1214.997,108.409,-49.314,-178.488,5.739,148.563
C00618=1214.992,108.658,-49.332,-178.485,5.740,148.562
C00619=1214.987,108.908,-49.352,-178.482,5.741,148.562
C00620=1214.983,109.156,-49.371,-178.480,5.741,148.561
C00621=1214.978,109.406,-49.390,-178.477,5.743,148.561
C00622=1214.972,109.655,-49.409,-178.474,5.744,148.560
C00623=1214.968,109.904,-49.428,-178.472,5.745,148.559
C00624=1214.963,110.153,-49.447,-178.469,5.746,148.559
C00625=1214.959,110.402,-49.466,-178.467,5.747,148.558
C00626=1214.953,110.651,-49.485,-178.464,5.748,148.558
C00627=1214.949,110.901,-49.505,-178.462,5.750,148.557
C00628=1214.944,111.149,-49.524,-178.459,5.750,148.557
C00629=1214.939,111.400,-49.543,-178.457,5.751,148.556
C00630=1214.934,111.649,-49.562,-178.454,5.753,148.556
C00631=1214.930,111.898,-49.581,-178.451,5.753,148.555
C00632=1214.924,112.147,-49.600,-178.449,5.754,148.555
C00633=1214.920,112.396,-49.620,-178.446,5.756,148.554
C00634=1214.916,112.645,-49.639,-178.444,5.756,148.554
C00635=1214.910,112.894,-49.658,-178.441,5.757,148.553
C00636=1214.905,113.144,-49.678,-178.438,5.759,148.553
C00637=1214.901,113.392,-49.697,-178.436,5.759,148.552
C00638=1214.896,113.642,-49.716,-178.434,5.760,148.552
C00639=1214.891,113.891,-49.736,-178.430,5.762,148.551
C00640=1214.886,114.140,-49.755,-178.428,5.763,148.550
C00641=1214.882,114.390,-49.774,-178.426,5.763,148.550
C00642=1214.877,114.639,-49.794,-178.423,5.765,148.549
C00643=1214.872,114.888,-49.813,-178.420,5.766,148.549
C00644=1214.867,115.137,-49.833,-178.418,5.766,148.548
C00645=1214.863,115.386,-49.852,-178.415,5.768,148.548
C00646=1214.858,115.636,-49.871,-178.412,5.769,148.547
C00647=1214.853,115.885,-49.891,-178.410,5.770,148.547
C00648=1214.848,116.134,-49.910,-178.407,5.771,148.546
C00649=1214.842,116.383,-49.930,-178.405,5.772,148.546
C00650=1214.838,116.632,-49.949,-178.402,5.774,148.545
C00651=1214.834,116.882,-49.968,-178.400,5.775,148.545
C00652=1214.828,117.131,-49.988,-178.397,5.775,148.544
C00653=1214.824,117.380,-50.007,-178.394,5.777,148.544
C00654=1214.818,117.629,-50.027,-178.392,5.778,148.543
C00655=1214.814,117.879,-50.046,-178.390,5.778,148.543
C00656=1214.810,118.128,-50.065,-178.387,5.780,148.542
C00657=1214.804,118.376,-50.085,-178.384,5.781,148.542
C00658=1214.800,118.626,-50.105,-178.381,5.782,148.541
C00659=1214.795,118.876,-50.125,-178.379,5.783,148.541
C00660=1214.790,119.124,-50.144,-178.376,5.784,148.540
C00661=1214.786,119.374,-50.163,-178.374,5.786,148.539
C00662=1214.781,119.623,-50.183,-178.371,5.786,148.539
C00663=1214.776,119.871,-50.203,-178.369,5.787,148.538
C00664=1214.771,120.121,-50.222,-178.366,5.789,148.538
C00665=1214.766,120.371,-50.242,-178.364,5.790,148.537
C00666=1214.762,120.620,-50.262,-178.361,5.791,148.537
C00667=1214.756,120.869,-50.281,-178.358,5.792,148.536
C00668=1214.752,121.118,-50.301,-178.356,5.793,148.536
C00669=1214.747,121.368,-50.321,-178.353,5.794,148.535
C00670=1214.742,121.616,-50.340,-178.351,5.795,148.535
C00671=1214.738,121.866,-50.359,-178.348,5.797,148.534
C00672=1214.733,122.115,-50.380,-178.345,5.797,148.534
C00673=1214.728,122.363,-50.399,-178.343,5.798,148.533
C00674=1214.723,122.613,-50.419,-178.340,5.800,148.533
C00675=1214.719,122.862,-50.439,-178.338,5.801,148.532
C00676=1214.714,123.112,-50.459,-178.335,5.802,148.532
C00677=1214.709,123.360,-50.478,-178.333,5.803,148.531
C00678=1214.704,123.609,-50.498,-178.330,5.804,148.531
C00679=1214.700,123.859,-50.518,-178.327,5.806,148.530
C00680=1214.695,124.109,-50.538,-178.325,5.806,148.530
C00681=1214.690,124.357,-50.558,-178.322,5.808,148.529
C00682=1214.685,124.606,-50.577,-178.319,5.809,148.529
C00683=1214.680,124.856,-50.597,-178.317,5.810,148.528
C00684=1214.676,125.105,-50.617,-178.315,5.811,148.528
C00685=1214.670,125.354,-50.637,-178.312,5.812,148.527
C00686=1214.666,125.603,-50.657,-178.309,5.814,148.527
C00687=1214.661,125.852,-50.677,-178.307,5.814,148.526
C00688=1214.657,126.101,-50.697,-178.304,5.816,148.526
C00689=1214.652,126.351,-50.717,-178.301,5.817,148.525
C00690=1214.647,126.600,-50.736,-178.299,5.818,148.525
C00691=1214.642,126.849,-50.756,-178.296,5.819,148.524
C00692=1214.638,127.098,-50.776,-178.294,5.820,148.524
C00693=1214.633,127.347,-50.796,-178.291,5.822,148.523
C00694=1214.628,127.597,-50.817,-178.289,5.823,148.523
C00695=1214.623,127.845,-50.837,-178.286,5.824,148.522
C00696=1214.618,128.095,-50.856,-178.283,5.825,148.522
C00697=1214.613,128.344,-50.877,-178.281,5.826,148.521
C00698=1214.609,128.593,-50.896,-178.278,5.827,148.521
C00699=1214.604,128.842,-50.917,-178.276,5.828,148.520
C00700=1214.600,129.092,-50.936,-178.273,5.830,148.519
C00701=1214.595,129.340,-50.956,-178.271,5.831,148.519
C00702=1214.590,129.589,-50.977,-178.268,5.832,148.518
C00703=1214.585,129.839,-50.996,-178.265,5.833,148.518
C00704=1214.580,130.088,-51.017,-178.262,5.835,148.517
C00705=1214.575,130.337,-51.037,-178.260,5.835,148.517
C00706=1214.571,130.586,-51.057,-178.258,5.836,148.517
C00707=1214.566,130.835,-51.077,-178.255,5.838,148.516
C00708=1214.561,131.084,-51.097,-178.253,5.839,148.516
C00709=1214.557,131.333,-51.117,-178.250,5.840,148.515
C00710=1214.551,131.583,-51.138,-178.247,5.841,148.515
C00711=1214.547,131.832,-51.158,-178.244,5.843,148.514
C00712=1214.542,132.081,-51.178,-178.242,5.844,148.514
C00713=1214.538,132.330,-51.198,-178.239,5.845,148.513
C00714=1214.533,132.579,-51.218,-178.237,5.846,148.513
C00715=1214.528,132.829,-51.239,-178.234,5.848,148.512
C00716=1214.523,133.097,-51.260,-178.232,5.849,148.512
C00717=1214.518,133.366,-51.283,-178.228,5.850,148.511
C00718=1214.512,133.635,-51.304,-178.226,5.852,148.511
C00719=1214.508,133.903,-51.326,-178.223,5.852,148.510
C00720=1214.503,134.152,-51.347,-178.221,5.854,148.510
C00721=1214.498,134.401,-51.367,-178.218,5.855,148.509
C00722=1214.493,134.650,-51.387,-178.215,5.857,148.509
C00723=1214.489,134.899,-51.408,-178.213,5.857,148.508
C00724=1214.484,135.149,-51.429,-178.210,5.859,148.508
C00725=1214.479,135.398,-51.448,-178.208,5.860,148.507
C00726=1214.474,135.647,-51.469,-178.205,5.861,148.506
C00727=1214.470,135.896,-51.489,-178.203,5.862,148.506
C00728=1214.465,136.145,-51.510,-178.199,5.864,148.505
C00729=1214.460,136.394,-51.530,-178.197,5.865,148.505
C00730=1214.455,136.643,-51.550,-178.195,5.867,148.505
C00731=1214.450,136.892,-51.571,-178.192,5.867,148.504
C00732=1214.445,137.141,-51.591,-178.190,5.868,148.504
C00733=1214.441,137.390,-51.611,-178.187,5.870,148.503
C00734=1214.436,137.640,-51.632,-178.185,5.871,148.503
C00735=1214.431,137.889,-51.653,-178.182,5.872,148.502
C00736=1214.427,138.137,-51.673,-178.179,5.873,148.502
C00737=1214.422,138.387,-51.694,-178.177,5.875,148.501
C00738=1214.417,138.636,-51.714,-178.174,5.875,148.501
C00739=1214.412,138.886,-51.735,-178.171,5.877,148.500
C00740=1214.407,139.135,-51.755,-178.169,5.878,148.500
C00741=1214.403,139.383,-51.775,-178.166,5.880,148.499
C00742=1214.398,139.633,-51.796,-178.164,5.881,148.499
C00743=1214.393,139.882,-51.817,-178.161,5.882,148.498
C00744=1214.388,140.131,-51.838,-178.158,5.884,148.498
C00745=1214.384,140.380,-51.858,-178.156,5.885,148.497
C00746=1214.379,140.629,-51.878,-178.153,5.886,148.497
C00747=1214.374,140.878,-51.899,-178.151,5.887,148.496
C00748=1214.370,141.127,-51.920,-178.148,5.889,148.496
C00749=1214.364,141.376,-51.941,-178.145,5.890,148.495
C00750=1214.361,141.626,-51.961,-178.143,5.891,148.495
C00751=1214.355,141.875,-51.982,-178.140,5.892,148.494
C00752=1214.351,142.124,-52.003,-178.138,5.894,148.494
C00753=1214.346,142.373,-52.025,-178.135,5.895,148.494
C00754=1214.342,142.622,-52.045,-178.132,5.896,148.493
C00755=1214.337,142.871,-52.065,-178.130,5.897,148.493
C00756=1214.332,143.120,-52.086,-178.127,5.899,148.492
C00757=1214.328,143.369,-52.107,-178.125,5.900,148.492
C00758=1214.322,143.618,-52.128,-178.122,5.902,148.491
C00759=1214.318,143.867,-52.148,-178.120,5.902,148.491
C00760=1214.313,144.116,-52.169,-178.117,5.904,148.490
C00761=1214.308,144.365,-52.189,-178.115,5.905,148.490
C00762=1214.304,144.614,-52.211,-178.112,5.906,148.489
C00763=1214.299,144.864,-52.232,-178.110,5.907,148.489
C00764=1214.295,145.113,-52.253,-178.107,5.909,148.488
C00765=1214.289,145.362,-52.274,-178.104,5.911,148.488
C00766=1214.285,145.611,-52.294,-178.102,5.912,148.487
C00767=1214.280,145.860,-52.316,-178.099,5.913,148.487
C00768=1214.276,146.109,-52.336,-178.096,5.914,148.486
C00769=1214.270,146.358,-52.357,-178.094,5.916,148.486
C00770=1214.266,146.607,-52.377,-178.092,5.917,148.486
C00771=1214.261,146.857,-52.399,-178.088,5.918,148.485
C00772=1214.257,147.106,-52.420,-178.086,5.919,148.485
C00773=1214.252,147.354,-52.441,-178.083,5.921,148.484
C00774=1214.247,147.604,-52.462,-178.081,5.922,148.484
C00775=1214.242,147.853,-52.483,-178.078,5.923,148.483
C00776=1214.238,148.101,-52.504,-178.075,5.925,148.483
C00777=1214.232,148.351,-52.525,-178.073,5.926,148.482
C00778=1214.229,148.600,-52.546,-178.070,5.928,148.482
C00779=1214.224,148.849,-52.567,-178.068,5.928,148.481
C00780=1214.219,149.098,-52.588,-178.065,5.930,148.481
C00781=1214.214,149.347,-52.609,-178.063,5.931,148.481
C00782=1214.209,149.596,-52.630,-178.060,5.933,148.480
C00783=1214.204,149.845,-52.651,-178.057,5.934,148.480
C00784=1214.200,150.095,-52.672,-178.055,5.935,148.479
C00785=1214.195,150.343,-52.694,-178.052,5.937,148.479
C00786=1214.190,150.593,-52.715,-178.050,5.938,148.478
C00787=1214.185,150.841,-52.736,-178.047,5.940,148.478
C00788=1214.181,151.090,-52.757,-178.045,5.941,148.477
C00789=1214.177,151.339,-52.779,-178.042,5.942,148.477
C00790=1214.172,151.589,-52.800,-178.039,5.944,148.476
C00791=1214.167,151.838,-52.820,-178.037,5.945,148.476
C00792=1214.162,152.086,-52.842,-178.034,5.946,148.475
C00793=1214.158,152.336,-52.863,-178.032,5.947,148.475
C00794=1214.153,152.585,-52.885,-178.029,5.949,148.475
C00795=1214.148,152.834,-52.905,-178.026,5.950,148.474
C00796=1214.143,153.082,-52.927,-178.024,5.951,148.474
C00797=1214.138,153.332,-52.948,-178.021,5.953,148.473
C00798=1214.134,153.581,-52.970,-178.019,5.954,148.473
C00799=1214.129,153.830,-52.991,-178.016,5.956,148.472
C00800=1214.125,154.079,-53.012,-178.014,5.957,148.472
C00801=1214.120,154.328,-53.033,-178.011,5.958,148.471
C00802=1214.115,154.577,-53.055,-178.008,5.960,148.471
C00803=1214.110,154.827,-53.076,-178.006,5.961,148.471
C00804=1214.105,155.075,-53.097,-178.003,5.963,148.470
C00805=1214.102,155.324,-53.119,-178.001,5.963,148.470
C00806=1214.097,155.573,-53.140,-177.998,5.965,148.469
C00807=1214.092,155.822,-53.162,-177.995,5.967,148.469
C00808=1214.086,156.071,-53.183,-177.993,5.968,148.468
C00809=1214.082,156.321,-53.205,-177.990,5.969,148.468
C00810=1214.077,156.569,-53.226,-177.987,5.971,148.467
C00811=1214.073,156.818,-53.247,-177.985,5.972,148.467
C00812=1214.069,157.068,-53.269,-177.982,5.974,148.466
C00813=1214.064,157.316,-53.290,-177.980,5.975,148.466
C00814=1214.059,157.566,-53.311,-177.977,5.976,148.466
C00815=1214.054,157.815,-53.333,-177.974,5.978,148.465
C00816=1214.049,158.064,-53.355,-177.972,5.979,148.465
C00817=1214.044,158.313,-53.376,-177.969,5.981,148.464
C00818=1214.040,158.562,-53.398,-177.967,5.982,148.464
C00819=1214.035,158.811,-53.420,-177.964,5.983,148.463
C00820=1214.030,159.080,-53.443,-177.962,5.985,148.463
C00821=1214.025,159.349,-53.466,-177.958,5.986,148.462
C00822=1214.020,159.618,-53.489,-177.956,5.988,148.462
C00823=1214.015,159.887,-53.513,-177.953,5.989,148.461
C00824=1214.010,160.136,-53.534,-177.950,5.991,148.461
C00825=1214.006,160.385,-53.556,-177.948,5.993,148.461
C00826=1214.001,160.634,-53.577,-177.946,5.994,148.460
C00827=1213.996,160.883,-53.599,-177.943,5.995,148.460
C00828=1213.992,161.132,-53.621,-177.940,5.997,148.459
C00829=1213.987,161.381,-53.643,-177.938,5.998,148.459
C00830=1213.982,161.630,-53.665,-177.935,6.000,148.459
C00831=1213.978,161.879,-53.687,-177.932,6.001,148.458
C00832=1213.972,162.128,-53.708,-177.930,6.002,148.458
C00833=1213.968,162.377,-53.730,-177.927,6.004,148.457
C00834=1213.963,162.626,-53.751,-177.925,6.006,148.457
C00835=1213.959,162.875,-53.773,-177.922,6.006,148.456
C00836=1213.954,163.124,-53.795,-177.919,6.008,148.456
C00837=1213.949,163.373,-53.817,-177.917,6.010,148.455
C00838=1213.945,163.622,-53.839,-177.915,6.011,148.455
C00839=1213.940,163.871,-53.860,-177.911,6.012,148.454
C00840=1213.936,164.120,-53.882,-177.909,6.013,148.454
C00841=1213.931,164.369,-53.904,-177.907,6.015,148.454
C00842=1213.927,164.618,-53.926,-177.904,6.017,148.453
C00843=1213.922,164.867,-53.948,-177.901,6.018,148.453
C00844=1213.918,165.116,-53.970,-177.899,6.019,148.452
C00845=1213.912,165.365,-53.992,-177.896,6.021,148.452
C00846=1213.907,165.614,-54.014,-177.894,6.022,148.452
C00847=1213.903,165.863,-54.036,-177.891,6.024,148.451
C00848=1213.898,166.112,-54.058,-177.888,6.026,148.451
C00849=1213.894,166.361,-54.080,-177.885,6.027,148.450
C00850=1213.889,166.609,-54.101,-177.883,6.028,148.450
C00851=1213.884,166.859,-54.123,-177.881,6.030,148.450
C00852=1213.880,167.107,-54.145,-177.878,6.032,148.449
C00853=1213.875,167.357,-54.168,-177.875,6.033,148.449
C00854=1213.870,167.606,-54.189,-177.873,6.034,148.448
C00855=1213.865,167.855,-54.211,-177.870,6.036,148.448
C00856=1213.861,168.104,-54.233,-177.868,6.037,148.447
C00857=1213.856,168.353,-54.255,-177.865,6.039,148.447
C00858=1213.851,168.602,-54.277,-177.862,6.040,148.447
C00859=1213.847,168.851,-54.300,-177.860,6.041,148.446
C00860=1213.842,169.099,-54.322,-177.857,6.043,148.446
C00861=1213.838,169.349,-54.344,-177.854,6.045,148.445
C00862=1213.833,169.597,-54.366,-177.852,6.046,148.445
C00863=1213.828,169.847,-54.388,-177.850,6.048,148.444
C00864=1213.823,170.096,-54.410,-177.847,6.049,148.444
C00865=1213.819,170.344,-54.433,-177.844,6.051,148.444
C00866=1213.815,170.594,-54.455,-177.842,6.052,148.443
C00867=1213.809,170.843,-54.477,-177.839,6.054,148.443
C00868=1213.805,171.092,-54.499,-177.836,6.055,148.442
C00869=1213.800,171.341,-54.521,-177.834,6.056,148.442
C00870=1213.796,171.589,-54.544,-177.832,6.058,148.442
C00871=1213.790,171.838,-54.566,-177.828,6.060,148.441
C00872=1213.786,172.088,-54.588,-177.826,6.061,148.441
C00873=1213.781,172.336,-54.610,-177.824,6.063,148.440
C00874=1213.777,172.585,-54.633,-177.821,6.064,148.440
C00875=1213.772,172.835,-54.655,-177.818,6.066,148.440
C00876=1213.767,173.083,-54.677,-177.816,6.067,148.439
C00877=1213.763,173.332,-54.699,-177.813,6.069,148.439
C00878=1213.758,173.581,-54.722,-177.810,6.070,148.438
C00879=1213.754,173.830,-54.744,-177.808,6.072,148.438
C00880=1213.750,174.079,-54.767,-177.806,6.073,148.437
C00881=1213.744,174.328,-54.789,-177.803,6.075,148.437
C00882=1213.740,174.577,-54.811,-177.800,6.077,148.437
C00883=1213.734,174.826,-54.834,-177.798,6.078,148.436
C00884=1213.730,175.075,-54.856,-177.795,6.079,148.436
C00885=1213.726,175.324,-54.879,-177.792,6.081,148.435
C00886=1213.721,175.573,-54.901,-177.790,6.083,148.435
C00887=1213.716,175.822,-54.923,-177.788,6.084,148.435
C00888=1213.712,176.071,-54.946,-177.785,6.086,148.434
C00889=1213.707,176.320,-54.968,-177.782,6.087,148.434
C00890=1213.703,176.568,-54.991,-177.779,6.089,148.433
C00891=1213.698,176.818,-55.013,-177.777,6.090,148.433
C00892=1213.693,177.066,-55.036,-177.774,6.092,148.433
C00893=1213.688,177.316,-55.058,-177.772,6.094,148.432
C00894=1213.684,177.564,-55.081,-177.769,6.095,148.432
C00895=1213.679,177.813,-55.103,-177.767,6.096,148.431
C00896=1213.675,178.062,-55.126,-177.764,6.098,148.431
C00897=1213.670,178.312,-55.148,-177.761,6.100,148.431
C00898=1213.665,178.560,-55.171,-177.759,6.102,148.430
C00899=1213.661,178.809,-55.193,-177.757,6.103,148.430
C00900=1213.656,179.058,-55.217,-177.754,6.105,148.430
C00901=1213.651,179.307,-55.238,-177.751,6.106,148.429
C00902=1213.647,179.556,-55.262,-177.748,6.108,148.429
C00903=1213.643,179.805,-55.285,-177.746,6.109,148.428
C00904=1213.638,180.054,-55.307,-177.743,6.111,148.428
C00905=1213.633,180.302,-55.330,-177.741,6.112,148.427
C00906=1213.628,180.551,-55.353,-177.738,6.114,148.427
C00907=1213.624,180.801,-55.375,-177.736,6.115,148.427
C00908=1213.619,181.049,-55.398,-177.733,6.117,148.426
C00909=1213.614,181.299,-55.421,-177.730,6.119,148.426
C00910=1213.610,181.547,-55.443,-177.727,6.120,148.425
C00911=1213.605,181.796,-55.467,-177.725,6.122,148.425
C00912=1213.600,182.045,-55.488,-177.723,6.123,148.425
C00913=1213.596,182.294,-55.512,-177.720,6.125,148.424
C00914=1213.592,182.543,-55.535,-177.717,6.127,148.424
C00915=1213.587,182.792,-55.558,-177.715,6.129,148.424
C00916=1213.581,183.041,-55.580,-177.712,6.129,148.423
C00917=1213.577,183.289,-55.603,-177.709,6.131,148.423
C00918=1213.573,183.539,-55.626,-177.707,6.133,148.422
C00919=1213.569,183.787,-55.649,-177.704,6.135,148.422
C00920=1213.564,184.037,-55.672,-177.702,6.137,148.422
C00921=1213.558,184.285,-55.695,-177.699,6.138,148.421
C00922=1213.554,184.534,-55.717,-177.697,6.139,148.421
C00923=1213.550,184.783,-55.741,-177.694,6.141,148.421
C00924=1213.545,185.052,-55.765,-177.691,6.143,148.420
C00925=1213.540,185.322,-55.790,-177.688,6.145,148.420
C00926=1213.534,185.592,-55.815,-177.686,6.146,148.419
C00927=1213.530,185.861,-55.840,-177.683,6.148,148.419
C00928=1213.525,186.110,-55.863,-177.680,6.150,148.418
C00929=1213.520,186.359,-55.886,-177.677,6.152,148.418
C00930=1213.516,186.607,-55.909,-177.675,6.153,148.418
C00931=1213.511,186.857,-55.932,-177.673,6.154,148.417
C00932=1213.506,187.106,-55.955,-177.670,6.156,148.417
C00933=1213.501,187.355,-55.978,-177.667,6.158,148.417
C00934=1213.498,187.604,-56.001,-177.665,6.160,148.416
C00935=1213.493,187.853,-56.024,-177.662,6.162,148.416
C00936=1213.488,188.102,-56.048,-177.660,6.163,148.415
C00937=1213.483,188.350,-56.071,-177.657,6.165,148.415
C00938=1213.479,188.599,-56.093,-177.654,6.166,148.415
C00939=1213.474,188.848,-56.117,-177.651,6.168,148.414
C00940=1213.469,189.097,-56.140,-177.649,6.170,148.414
C00941=1213.465,189.346,-56.164,-177.647,6.171,148.413
C00942=1213.461,189.595,-56.186,-177.644,6.172,148.413
C00943=1213.456,189.844,-56.210,-177.641,6.174,148.413
C00944=1213.451,190.093,-56.233,-177.639,6.176,148.412
C00945=1213.446,190.341,-56.256,-177.636,6.178,148.412
C00946=1213.441,190.590,-56.279,-177.633,6.180,148.412
C00947=1213.437,190.839,-56.302,-177.631,6.181,148.411
C00948=1213.433,191.088,-56.326,-177.629,6.183,148.411
C00949=1213.428,191.337,-56.349,-177.626,6.184,148.411
C00950=1213.423,191.586,-56.372,-177.623,6.186,148.410
C00951=1213.419,191.835,-56.396,-177.620,6.188,148.410
C00952=1213.414,192.084,-56.420,-177.618,6.190,148.409
C00953=1213.410,192.333,-56.443,-177.615,6.191,148.409
C00954=1213.406,192.581,-56.466,-177.613,6.192,148.409
C00955=1213.401,192.830,-56.489,-177.610,6.194,148.408
C00956=1213.396,193.079,-56.513,-177.608,6.196,148.408
C00957=1213.391,193.328,-56.536,-177.605,6.198,148.408
C00958=1213.386,193.577,-56.559,-177.602,6.200,148.407
C00959=1213.382,193.825,-56.583,-177.600,6.202,148.407
C00960=1213.377,194.074,-56.606,-177.597,6.203,148.407
C00961=1213.372,194.323,-56.630,-177.595,6.204,148.406
C00962=1213.368,194.572,-56.653,-177.592,6.206,148.406
C00963=1213.363,194.821,-56.677,-177.590,6.208,148.405
C00964=1213.359,195.070,-56.700,-177.587,6.210,148.405
C00965=1213.354,195.319,-56.724,-177.584,6.212,148.405
C00966=1213.350,195.567,-56.747,-177.582,6.214,148.404
C00967=1213.346,195.816,-56.771,-177.579,6.215,148.404
C00968=1213.341,196.065,-56.794,-177.577,6.216,148.404
C00969=1213.336,196.314,-56.817,-177.574,6.218,148.403
C00970=1213.331,196.563,-56.841,-177.572,6.220,148.403
C00971=1213.327,196.811,-56.865,-177.569,6.222,148.403
C00972=1213.322,197.060,-56.888,-177.566,6.223,148.402
C00973=1213.318,197.309,-56.912,-177.563,6.225,148.402
C00974=1213.313,197.558,-56.936,-177.560,6.227,148.401
C00975=1213.309,197.807,-56.959,-177.558,6.229,148.401
C00976=1213.304,198.056,-56.982,-177.556,6.230,148.401
C00977=1213.299,198.304,-57.006,-177.553,6.232,148.400
C00978=1213.294,198.554,-57.030,-177.550,6.234,148.400
C00979=1213.290,198.803,-57.055,-177.548,6.235,148.400
C00980=1213.286,199.052,-57.078,-177.545,6.237,148.399
C00981=1213.281,199.301,-57.101,-177.543,6.239,148.399
C00982=1213.276,199.549,-57.126,-177.540,6.241,148.399
C00983=1213.272,199.798,-57.149,-177.537,6.243,148.398
C00984=1213.267,200.047,-57.173,-177.535,6.245,148.398
C00985=1213.263,200.296,-57.196,-177.532,6.246,148.398
C00986=1213.258,200.544,-57.220,-177.530,6.247,148.397
C00987=1213.254,200.793,-57.244,-177.527,6.249,148.397
C00988=1213.249,201.042,-57.268,-177.525,6.251,148.397
C00989=1213.244,201.291,-57.291,-177.522,6.253,148.396
C00990=1213.239,201.539,-57.316,-177.519,6.255,148.396
C00991=1213.235,201.788,-57.339,-177.517,6.257,148.396
C00992=1213.231,202.038,-57.364,-177.514,6.258,148.395
C00993=1213.226,202.287,-57.387,-177.511,6.260,148.395
C00994=1213.222,202.535,-57.411,-177.509,6.262,148.395
C00995=1213.217,202.783,-57.435,-177.506,6.264,148.394
C00996=1213.212,203.033,-57.459,-177.504,6.265,148.394
C00997=1213.208,203.281,-57.483,-177.501,6.267,148.393
C00998=1213.203,203.530,-57.507,-177.499,6.269,148.393
C00999=1213.198,203.779,-57.531,-177.496,6.270,148.393
C01000=1213.195,204.028,-57.555,-177.493,6.272,148.392
C01001=1213.190,204.277,-57.578,-177.491,6.274,148.392
C01002=1213.185,204.525,-57.603,-177.488,6.276,148.392
C01003=1213.180,204.774,-57.626,-177.485,6.278,148.391
C01004=1213.176,205.023,-57.651,-177.483,6.280,148.391
C01005=1213.171,205.271,-57.675,-177.480,6.281,148.391
C01006=1213.167,205.521,-57.700,-177.478,6.283,148.390
C01007=1213.162,205.770,-57.723,-177.475,6.285,148.390
C01008=1213.158,206.018,-57.747,-177.472,6.287,148.390
C01009=1213.153,206.267,-57.771,-177.470,6.288,148.389
C01010=1213.148,206.516,-57.795,-177.468,6.290,148.389
C01011=1213.143,206.764,-57.819,-177.465,6.292,148.389
C01012=1213.140,207.013,-57.844,-177.463,6.294,148.389
C01013=1213.135,207.262,-57.868,-177.460,6.296,148.388
C01014=1213.130,207.511,-57.892,-177.457,6.297,148.388
C01015=1213.125,207.760,-57.916,-177.455,6.299,148.388
C01016=1213.121,208.008,-57.940,-177.452,6.301,148.387
C01017=1213.117,208.257,-57.965,-177.450,6.303,148.387
C01018=1213.112,208.506,-57.989,-177.447,6.305,148.387
C01019=1213.107,208.755,-58.014,-177.444,6.307,148.386
C01020=1213.102,209.004,-58.037,-177.442,6.309,148.386
C01021=1213.098,209.253,-58.061,-177.439,6.310,148.386
C01022=1213.093,209.501,-58.086,-177.436,6.312,148.385
C01023=1213.089,209.750,-58.110,-177.434,6.314,148.385
C01024=1213.085,209.998,-58.134,-177.431,6.316,148.385
C01025=1213.080,210.248,-58.159,-177.428,6.318,148.384
C01026=1213.076,210.496,-58.183,-177.426,6.320,148.384
C01027=1213.071,210.745,-58.208,-177.423,6.321,148.384
C01028=1213.066,211.015,-58.233,-177.420,6.323,148.383
C01029=1213.061,211.286,-58.260,-177.418,6.325,148.383
C01030=1213.056,211.556,-58.287,-177.415,6.327,148.383
C01031=1213.051,211.827,-58.314,-177.412,6.330,148.382
C01032=1213.047,212.075,-58.338,-177.409,6.331,148.382
C01033=1213.042,212.324,-58.363,-177.407,6.333,148.382
C01034=1213.038,212.573,-58.387,-177.404,6.335,148.381
C01035=1213.032,212.821,-58.412,-177.401,6.337,148.381
C01036=1213.028,213.070,-58.436,-177.399,6.339,148.381
C01037=1213.024,213.319,-58.461,-177.397,6.340,148.380
C01038=1213.019,213.568,-58.485,-177.394,6.342,148.380
C01039=1213.015,213.816,-58.509,-177.391,6.343,148.380
C01040=1213.010,214.066,-58.534,-177.389,6.346,148.379
C01041=1213.006,214.314,-58.558,-177.387,6.347,148.379
C01042=1213.001,214.563,-58.583,-177.384,6.349,148.379
C01043=1212.996,214.812,-58.608,-177.381,6.351,148.378
C01044=1212.992,215.061,-58.632,-177.379,6.353,148.378
C01045=1212.987,215.309,-58.657,-177.376,6.355,148.378
C01046=1212.983,215.558,-58.681,-177.373,6.357,148.377
C01047=1212.978,215.806,-58.706,-177.371,6.359,148.377
C01048=1212.974,216.055,-58.730,-177.368,6.360,148.377
C01049=1212.969,216.304,-58.756,-177.366,6.362,148.376
C01050=1212.965,216.553,-58.780,-177.363,6.364,148.376
C01051=1212.960,216.802,-58.805,-177.361,6.366,148.376
C01052=1212.955,217.050,-58.830,-177.358,6.368,148.376
C01053=1212.951,217.299,-58.854,-177.355,6.370,148.375
C01054=1212.946,217.548,-58.879,-177.353,6.372,148.375
C01055=1212.942,217.797,-58.903,-177.350,6.374,148.375
C01056=1212.938,218.046,-58.928,-177.347,6.376,148.374
C01057=1212.933,218.294,-58.954,-177.344,6.378,148.374
C01058=1212.928,218.542,-58.978,-177.342,6.380,148.374
C01059=1212.924,218.792,-59.003,-177.339,6.382,148.373
C01060=1212.920,219.040,-59.028,-177.336,6.384,148.373
C01061=1212.915,219.289,-59.053,-177.334,6.386,148.373
C01062=1212.910,219.538,-59.077,-177.332,6.388,148.373
C01063=1212.906,219.786,-59.101,-177.329,6.390,148.372
C01064=1212.901,220.035,-59.127,-177.326,6.391,148.372
C01065=1212.896,220.284,-59.152,-177.324,6.393,148.372
C01066=1212.893,220.532,-59.177,-177.321,6.395,148.371
C01067=1212.888,220.781,-59.202,-177.318,6.397,148.371
C01068=1212.883,221.030,-59.227,-177.316,6.399,148.371
C01069=1212.878,221.279,-59.252,-177.314,6.401,148.370
C01070=1212.875,221.528,-59.276,-177.311,6.403,148.370
C01071=1212.869,221.776,-59.301,-177.308,6.405,148.370
C01072=1212.865,222.025,-59.327,-177.306,6.406,148.370
C01073=1212.861,222.274,-59.351,-177.303,6.408,148.369
C01074=1212.857,222.522,-59.377,-177.301,6.410,148.369
C01075=1212.851,222.771,-59.401,-177.298,6.412,148.369
C01076=1212.847,223.019,-59.427,-177.296,6.414,148.368
C01077=1212.843,223.268,-59.451,-177.293,6.416,148.368
C01078=1212.838,223.516,-59.477,-177.290,6.418,148.368
C01079=1212.833,223.766,-59.502,-177.288,6.420,148.367
C01080=1212.829,224.014,-59.527,-177.285,6.422,148.367
C01081=1212.824,224.263,-59.552,-177.283,6.423,148.367
C01082=1212.820,224.511,-59.577,-177.280,6.426,148.367
C01083=1212.815,224.761,-59.602,-177.278,6.427,148.366
C01084=1212.811,225.009,-59.628,-177.275,6.429,148.366
C01085=1212.806,225.258,-59.652,-177.273,6.431,148.366
C01086=1212.802,225.507,-59.678,-177.270,6.433,148.365
C01087=1212.797,225.755,-59.703,-177.267,6.435,148.365
C01088=1212.793,226.004,-59.728,-177.265,6.437,148.365
C01089=1212.788,226.252,-59.753,-177.262,6.439,148.365
C01090=1212.784,226.502,-59.778,-177.259,6.442,148.364
C01091=1212.779,226.750,-59.804,-177.257,6.443,148.364
C01092=1212.775,226.999,-59.829,-177.254,6.445,148.364
C01093=1212.770,227.247,-59.854,-177.252,6.447,148.364
C01094=1212.765,227.496,-59.880,-177.249,6.449,148.363
C01095=1212.761,227.745,-59.906,-177.247,6.451,148.363
C01096=1212.756,227.994,-59.930,-177.244,6.453,148.363
C01097=1212.753,228.242,-59.955,-177.241,6.455,148.362
C01098=1212.748,228.490,-59.981,-177.239,6.457,148.362
C01099=1212.744,228.739,-60.006,-177.237,6.459,148.362
C01100=1212.739,228.988,-60.032,-177.234,6.461,148.362
C01101=1212.734,229.237,-60.057,-177.231,6.463,148.361
C01102=1212.730,229.485,-60.083,-177.229,6.464,148.361
C01103=1212.725,229.733,-60.108,-177.227,6.467,148.361
C01104=1212.721,229.983,-60.133,-177.224,6.468,148.360
C01105=1212.716,230.232,-60.159,-177.221,6.470,148.360
C01106=1212.712,230.480,-60.184,-177.219,6.472,148.360
C01107=1212.707,230.729,-60.210,-177.215,6.475,148.360
C01108=1212.703,230.977,-60.236,-177.213,6.477,148.359
C01109=1212.698,231.226,-60.260,-177.211,6.479,148.359
C01110=1212.694,231.475,-60.286,-177.208,6.481,148.359
C01111=1212.689,231.723,-60.312,-177.205,6.483,148.358
C01112=1212.685,231.972,-60.337,-177.203,6.485,148.358
C01113=1212.681,232.221,-60.363,-177.201,6.487,148.358
C01114=1212.676,232.469,-60.388,-177.198,6.488,148.358
C01115=1212.671,232.718,-60.414,-177.195,6.490,148.357
C01116=1212.667,232.966,-60.440,-177.193,6.492,148.357
C01117=1212.662,233.215,-60.465,-177.191,6.494,148.357
C01118=1212.658,233.464,-60.490,-177.188,6.496,148.357
C01119=1212.653,233.713,-60.517,-177.185,6.499,148.356
C01120=1212.648,233.961,-60.542,-177.182,6.501,148.356
C01121=1212.644,234.210,-60.568,-177.180,6.503,148.356
C01122=1212.640,234.459,-60.594,-177.177,6.505,148.356
C01123=1212.635,234.708,-60.619,-177.175,6.507,148.355
C01124=1212.631,234.956,-60.645,-177.172,6.508,148.355
C01125=1212.626,235.204,-60.670,-177.170,6.511,148.355
C01126=1212.622,235.453,-60.696,-177.167,6.512,148.355
C01127=1212.617,235.701,-60.722,-177.165,6.514,148.354
C01128=1212.612,235.950,-60.748,-177.163,6.517,148.354
C01129=1212.608,236.199,-60.774,-177.160,6.518,148.354
C01130=1212.604,236.448,-60.799,-177.157,6.521,148.354
C01131=1212.599,236.696,-60.826,-177.154,6.523,148.353
C01132=1212.595,236.967,-60.854,-177.152,6.525,148.353
C01133=1212.590,237.239,-60.882,-177.149,6.527,148.353
C01134=1212.585,237.510,-60.910,-177.146,6.530,148.353
C01135=1212.580,237.782,-60.939,-177.144,6.532,148.352
C01136=1212.575,238.031,-60.964,-177.141,6.533,148.352
C01137=1212.571,238.279,-60.990,-177.138,6.535,148.352
C01138=1212.566,238.528,-61.016,-177.136,6.538,148.352
C01139=1212.562,238.776,-61.042,-177.133,6.540,148.351
C01140=1212.557,239.025,-61.068,-177.130,6.542,148.351
C01141=1212.553,239.273,-61.094,-177.128,6.544,148.351
C01142=1212.548,239.522,-61.119,-177.126,6.546,148.350
C01143=1212.544,239.771,-61.145,-177.123,6.548,148.350
C01144=1212.540,240.019,-61.172,-177.120,6.550,148.350
C01145=1212.535,240.268,-61.198,-177.118,6.552,148.350
C01146=1212.530,240.516,-61.223,-177.115,6.555,148.349
C01147=1212.525,240.765,-61.250,-177.112,6.556,148.349
C01148=1212.522,241.014,-61.276,-177.110,6.559,148.349
C01149=1212.517,241.262,-61.302,-177.108,6.560,148.349
C01150=1212.513,241.511,-61.328,-177.105,6.562,148.348
C01151=1212.508,241.760,-61.355,-177.102,6.564,148.348
C01152=1212.504,242.008,-61.380,-177.100,6.566,148.348
C01153=1212.499,242.257,-61.406,-177.098,6.568,148.348
C01154=1212.495,242.505,-61.433,-177.094,6.571,148.347
C01155=1212.491,242.754,-61.459,-177.092,6.573,148.347
C01156=1212.486,243.003,-61.485,-177.090,6.575,148.347
C01157=1212.482,243.251,-61.512,-177.087,6.577,148.347
C01158=1212.477,243.500,-61.537,-177.085,6.579,148.347
C01159=1212.472,243.748,-61.564,-177.082,6.581,148.346
C01160=1212.468,243.997,-61.590,-177.080,6.583,148.346
C01161=1212.464,244.245,-61.615,-177.077,6.586,148.346
C01162=1212.459,244.494,-61.643,-177.074,6.588,148.346
C01163=1212.455,244.743,-61.668,-177.072,6.589,148.345
C01164=1212.450,244.991,-61.695,-177.070,6.592,148.345
C01165=1212.446,245.240,-61.721,-177.067,6.593,148.345
C01166=1212.441,245.488,-61.748,-177.064,6.595,148.345
C01167=1212.437,245.737,-61.774,-177.062,6.598,148.345
C01168=1212.433,245.985,-61.800,-177.059,6.600,148.344
C01169=1212.428,246.234,-61.826,-177.056,6.602,148.344
C01170=1212.424,246.482,-61.853,-177.054,6.604,148.344
C01171=1212.419,246.731,-61.879,-177.052,6.606,148.343
C01172=1212.415,246.979,-61.906,-177.049,6.608,148.343
C01173=1212.410,247.228,-61.932,-177.046,6.611,148.343
C01174=1212.406,247.477,-61.958,-177.044,6.613,148.343
C01175=1212.401,247.725,-61.986,-177.041,6.615,148.343
C01176=1212.397,247.974,-62.011,-177.039,6.617,148.342
C01177=1212.392,248.222,-62.038,-177.036,6.619,148.342
C01178=1212.388,248.471,-62.064,-177.034,6.621,148.342
C01179=1212.383,248.720,-62.091,-177.031,6.624,148.342
C01180=1212.380,248.968,-62.118,-177.028,6.625,148.341
C01181=1212.375,249.217,-62.144,-177.026,6.628,148.341
C01182=1212.370,249.466,-62.171,-177.024,6.630,148.341
C01183=1212.366,249.714,-62.197,-177.021,6.631,148.341
C01184=1212.361,249.963,-62.224,-177.019,6.634,148.341
C01185=1212.357,250.211,-62.250,-177.016,6.636,148.340
C01186=1212.352,250.460,-62.277,-177.013,6.638,148.340
C01187=1212.348,250.708,-62.303,-177.011,6.640,148.340
C01188=1212.344,250.957,-62.330,-177.008,6.642,148.340
C01189=1212.339,251.205,-62.357,-177.006,6.644,148.340
C01190=1212.335,251.454,-62.384,-177.003,6.647,148.339
C01191=1212.330,251.703,-62.410,-177.001,6.649,148.339
C01192=1212.326,251.951,-62.437,-176.998,6.651,148.339
C01193=1212.321,252.199,-62.464,-176.996,6.653,148.339
C01194=1212.317,252.448,-62.491,-176.993,6.655,148.338
C01195=1212.313,252.696,-62.517,-176.990,6.658,148.338
C01196=1212.308,252.945,-62.543,-176.988,6.660,148.338
C01197=1212.303,253.194,-62.571,-176.985,6.662,148.338
C01198=1212.299,253.442,-62.597,-176.983,6.664,148.338
C01199=1212.295,253.690,-62.624,-176.981,6.666,148.337
C01200=1212.290,253.939,-62.651,-176.978,6.669,148.337
C01201=1212.285,254.187,-62.678,-176.975,6.671,148.337
C01202=1212.281,254.435,-62.705,-176.973,6.673,148.337
C01203=1212.277,254.684,-62.732,-176.970,6.675,148.336
C01204=1212.272,254.933,-62.758,-176.967,6.678,148.336
C01205=1212.268,255.181,-62.785,-176.965,6.679,148.336
C01206=1212.263,255.430,-62.812,-176.963,6.682,148.336
C01207=1212.259,255.679,-62.839,-176.960,6.684,148.336
C01208=1212.255,255.927,-62.866,-176.958,6.686,148.336
C01209=1212.251,256.176,-62.893,-176.955,6.688,148.335
C01210=1212.246,256.424,-62.920,-176.952,6.690,148.335
C01211=1212.241,256.673,-62.947,-176.950,6.692,148.335
C01212=1212.237,256.921,-62.974,-176.947,6.694,148.335
C01213=1212.233,257.169,-63.000,-176.945,6.697,148.335
C01214=1212.228,257.418,-63.027,-176.942,6.699,148.334
C01215=1212.223,257.666,-63.054,-176.940,6.701,148.334
C01216=1212.219,257.916,-63.082,-176.937,6.703,148.334
C01217=1212.215,258.164,-63.109,-176.935,6.706,148.334
C01218=1212.210,258.412,-63.136,-176.932,6.708,148.334
C01219=1212.206,258.660,-63.163,-176.929,6.710,148.333
C01220=1212.202,258.909,-63.190,-176.927,6.712,148.333
C01221=1212.197,259.157,-63.217,-176.924,6.715,148.333
C01222=1212.193,259.406,-63.244,-176.922,6.717,148.333
C01223=1212.188,259.655,-63.272,-176.919,6.719,148.333
C01224=1212.184,259.903,-63.299,-176.917,6.721,148.332
C01225=1212.179,260.152,-63.326,-176.914,6.724,148.332
C01226=1212.176,260.399,-63.353,-176.912,6.726,148.332
C01227=1212.171,260.648,-63.380,-176.909,6.728,148.332
C01228=1212.166,260.896,-63.407,-176.907,6.730,148.332
C01229=1212.162,261.145,-63.434,-176.904,6.733,148.331
C01230=1212.158,261.394,-63.462,-176.902,6.735,148.331
C01231=1212.153,261.642,-63.489,-176.899,6.737,148.331
C01232=1212.148,261.890,-63.516,-176.897,6.739,148.331
C01233=1212.144,262.139,-63.543,-176.894,6.742,148.331
C01234=1212.140,262.388,-63.571,-176.892,6.744,148.331
C01235=1212.135,262.636,-63.599,-176.889,6.746,148.330
C01236=1212.131,262.909,-63.628,-176.886,6.748,148.330
C01237=1212.125,263.181,-63.658,-176.884,6.751,148.330
C01238=1212.121,263.454,-63.688,-176.881,6.753,148.330
C01239=1212.116,263.727,-63.718,-176.878,6.756,148.330
C01240=1212.111,263.976,-63.745,-176.875,6.758,148.329
C01241=1212.107,264.223,-63.773,-176.873,6.760,148.329
C01242=1212.102,264.472,-63.800,-176.871,6.762,148.329
C01243=1212.099,264.721,-63.828,-176.868,6.765,148.329
C01244=1212.094,264.969,-63.855,-176.865,6.767,148.329
C01245=1212.089,265.218,-63.883,-176.863,6.769,148.329
C01246=1212.086,265.466,-63.911,-176.860,6.772,148.328
C01247=1212.081,265.715,-63.938,-176.858,6.774,148.328
C01248=1212.077,265.962,-63.966,-176.855,6.776,148.328
C01249=1212.072,266.211,-63.993,-176.853,6.778,148.328
C01250=1212.068,266.460,-64.020,-176.850,6.781,148.328
C01251=1212.064,266.708,-64.048,-176.848,6.783,148.328
C01252=1212.058,266.957,-64.075,-176.845,6.785,148.327
C01253=1212.054,267.205,-64.104,-176.843,6.788,148.327
C01254=1212.050,267.454,-64.131,-176.840,6.790,148.327
C01255=1212.045,267.702,-64.158,-176.838,6.792,148.327
C01256=1212.041,267.950,-64.185,-176.835,6.795,148.327
C01257=1212.037,268.199,-64.214,-176.832,6.797,148.326
C01258=1212.032,268.447,-64.241,-176.830,6.799,148.326
C01259=1212.028,268.695,-64.268,-176.828,6.801,148.326
C01260=1212.024,268.944,-64.297,-176.825,6.804,148.326
C01261=1212.019,269.193,-64.324,-176.822,6.806,148.326
C01262=1212.015,269.441,-64.352,-176.820,6.808,148.326
C01263=1212.010,269.690,-64.379,-176.817,6.811,148.325
C01264=1212.006,269.938,-64.407,-176.815,6.813,148.325
C01265=1212.002,270.186,-64.435,-176.812,6.815,148.325
C01266=1211.997,270.435,-64.463,-176.810,6.818,148.325
C01267=1211.993,270.683,-64.491,-176.808,6.820,148.325
C01268=1211.989,270.931,-64.519,-176.805,6.822,148.325
C01269=1211.984,271.180,-64.546,-176.802,6.825,148.325
C01270=1211.979,271.428,-64.574,-176.800,6.827,148.324
C01271=1211.975,271.677,-64.603,-176.798,6.829,148.324
C01272=1211.971,271.925,-64.630,-176.795,6.832,148.324
C01273=1211.967,272.174,-64.658,-176.792,6.834,148.324
C01274=1211.962,272.422,-64.686,-176.790,6.836,148.324
C01275=1211.958,272.670,-64.714,-176.787,6.839,148.324
C01276=1211.953,272.919,-64.741,-176.785,6.841,148.324
C01277=1211.949,273.167,-64.769,-176.782,6.843,148.323
C01278=1211.945,273.416,-64.798,-176.779,6.846,148.323
C01279=1211.940,273.664,-64.826,-176.777,6.848,148.323
C01280=1211.936,273.912,-64.853,-176.775,6.850,148.323
C01281=1211.931,274.161,-64.881,-176.772,6.853,148.323
C01282=1211.927,274.409,-64.909,-176.770,6.855,148.323
C01283=1211.923,274.657,-64.937,-176.767,6.857,148.322
C01284=1211.918,274.906,-64.966,-176.765,6.860,148.322
C01285=1211.914,275.154,-64.994,-176.762,6.862,148.322
C01286=1211.910,275.402,-65.022,-176.759,6.865,148.322
C01287=1211.905,275.652,-65.050,-176.757,6.867,148.322
C01288=1211.901,275.900,-65.077,-176.755,6.869,148.322
C01289=1211.897,276.148,-65.106,-176.752,6.872,148.322
C01290=1211.892,276.396,-65.134,-176.749,6.874,148.321
C01291=1211.888,276.645,-65.162,-176.747,6.876,148.321
C01292=1211.883,276.893,-65.190,-176.744,6.879,148.321
C01293=1211.879,277.142,-65.219,-176.742,6.881,148.321
C01294=1211.875,277.389,-65.246,-176.740,6.883,148.321
C01295=1211.870,277.638,-65.275,-176.737,6.886,148.321
C01296=1211.866,277.886,-65.303,-176.734,6.888,148.321
C01297=1211.862,278.135,-65.332,-176.732,6.891,148.321
C01298=1211.857,278.383,-65.359,-176.730,6.894,148.320
C01299=1211.853,278.632,-65.388,-176.727,6.895,148.320
C01300=1211.848,278.880,-65.416,-176.724,6.898,148.320
C01301=1211.845,279.128,-65.444,-176.722,6.901,148.320
C01302=1211.840,279.377,-65.472,-176.720,6.903,148.320
C01303=1211.836,279.625,-65.501,-176.717,6.906,148.320
C01304=1211.831,279.873,-65.529,-176.715,6.908,148.320
C01305=1211.827,280.121,-65.558,-176.712,6.910,148.319
C01306=1211.822,280.369,-65.586,-176.709,6.913,148.319
C01307=1211.818,280.618,-65.614,-176.707,6.915,148.319
C01308=1211.814,280.867,-65.643,-176.704,6.918,148.319
C01309=1211.810,281.115,-65.671,-176.702,6.920,148.319
C01310=1211.805,281.364,-65.700,-176.699,6.923,148.319
C01311=1211.801,281.612,-65.727,-176.697,6.925,148.319
C01312=1211.797,281.860,-65.757,-176.695,6.927,148.319
C01313=1211.792,282.108,-65.785,-176.692,6.930,148.319
C01314=1211.788,282.357,-65.813,-176.690,6.932,148.318
C01315=1211.783,282.605,-65.842,-176.687,6.935,148.318
C01316=1211.779,282.853,-65.870,-176.685,6.937,148.318
C01317=1211.775,283.102,-65.899,-176.682,6.939,148.318
C01318=1211.770,283.350,-65.928,-176.679,6.942,148.318
C01319=1211.766,283.598,-65.956,-176.677,6.944,148.318
C01320=1211.761,283.847,-65.985,-176.674,6.947,148.318
C01321=1211.757,284.095,-66.013,-176.672,6.949,148.318
C01322=1211.753,284.343,-66.042,-176.670,6.951,148.317
C01323=1211.748,284.592,-66.070,-176.667,6.954,148.317
C01324=1211.744,284.840,-66.099,-176.665,6.956,148.317
C01325=1211.740,285.088,-66.128,-176.662,6.959,148.317
C01326=1211.735,285.337,-66.156,-176.660,6.961,148.317
C01327=1211.731,285.585,-66.185,-176.657,6.964,148.317
C01328=1211.727,285.833,-66.214,-176.655,6.967,148.317
C01329=1211.722,286.081,-66.243,-176.652,6.968,148.317
C01330=1211.718,286.330,-66.271,-176.650,6.972,148.317
C01331=1211.714,286.578,-66.300,-176.647,6.974,148.317
C01332=1211.709,286.826,-66.329,-176.645,6.977,148.317
C01333=1211.705,287.075,-66.357,-176.642,6.979,148.316
C01334=1211.701,287.323,-66.386,-176.640,6.981,148.316
C01335=1211.696,287.571,-66.415,-176.637,6.984,148.316
C01336=1211.692,287.819,-66.444,-176.635,6.986,148.316
C01337=1211.688,288.068,-66.472,-176.632,6.989,148.316
C01338=1211.683,288.315,-66.501,-176.630,6.991,148.316
C01339=1211.679,288.564,-66.530,-176.627,6.994,148.316
C01340=1211.674,288.839,-66.562,-176.625,6.996,148.316
C01341=1211.670,289.112,-66.594,-176.622,6.999,148.315
C01342=1211.665,289.387,-66.626,-176.619,7.002,148.315
C01343=1211.660,289.661,-66.657,-176.617,7.005,148.315
C01344=1211.656,289.909,-66.687,-176.614,7.007,148.315
C01345=1211.651,290.158,-66.716,-176.611,7.010,148.315
C01346=1211.646,290.406,-66.745,-176.609,7.012,148.315
C01347=1211.642,290.654,-66.774,-176.606,7.015,148.315
C01348=1211.638,290.903,-66.803,-176.604,7.017,148.315
C01349=1211.634,291.151,-66.832,-176.602,7.019,148.315
C01350=1211.629,291.399,-66.860,-176.599,7.022,148.315
C01351=1211.625,291.647,-66.890,-176.597,7.024,148.315
C01352=1211.621,291.896,-66.919,-176.594,7.027,148.315
C01353=1211.616,292.145,-66.948,-176.592,7.030,148.314
C01354=1211.612,292.393,-66.977,-176.589,7.033,148.314
C01355=1211.607,292.640,-67.006,-176.587,7.035,148.314
C01356=1211.604,292.888,-67.035,-176.584,7.038,148.314
C01357=1211.600,293.137,-67.064,-176.582,7.040,148.314
C01358=1211.595,293.386,-67.093,-176.579,7.043,148.314
C01359=1211.591,293.634,-67.123,-176.577,7.045,148.314
C01360=1211.586,293.881,-67.152,-176.575,7.047,148.314
C01361=1211.582,294.130,-67.181,-176.572,7.050,148.314
C01362=1211.578,294.379,-67.210,-176.570,7.052,148.314
C01363=1211.574,294.627,-67.240,-176.567,7.055,148.314
C01364=1211.569,294.875,-67.269,-176.565,7.057,148.314
C01365=1211.565,295.123,-67.298,-176.562,7.060,148.314
C01366=1211.560,295.372,-67.327,-176.560,7.063,148.313
C01367=1211.556,295.620,-67.356,-176.558,7.066,148.313
C01368=1211.552,295.868,-67.386,-176.555,7.068,148.313
C01369=1211.548,296.116,-67.415,-176.552,7.071,148.313
C01370=1211.543,296.365,-67.445,-176.550,7.073,148.313
C01371=1211.539,296.613,-67.474,-176.547,7.076,148.313
C01372=1211.534,296.860,-67.503,-176.545,7.078,148.313
C01373=1211.530,297.109,-67.533,-176.543,7.081,148.313
C01374=1211.526,297.357,-67.562,-176.540,7.083,148.313
C01375=1211.522,297.606,-67.591,-176.538,7.086,148.313
C01376=1211.517,297.854,-67.620,-176.536,7.088,148.313
C01377=1211.513,298.102,-67.650,-176.533,7.091,148.313
C01378=1211.509,298.351,-67.679,-176.531,7.094,148.313
C01379=1211.505,298.599,-67.709,-176.528,7.097,148.313
C01380=1211.501,298.847,-67.738,-176.526,7.099,148.313
C01381=1211.496,299.095,-67.767,-176.523,7.102,148.312
C01382=1211.492,299.343,-67.797,-176.521,7.104,148.312
C01383=1211.487,299.592,-67.827,-176.519,7.106,148.312
C01384=1211.483,299.839,-67.857,-176.516,7.109,148.312
C01385=1211.479,300.088,-67.886,-176.514,7.111,148.312
C01386=1211.475,300.336,-67.916,-176.511,7.114,148.312
C01387=1211.470,300.584,-67.945,-176.509,7.117,148.312
C01388=1211.466,300.832,-67.975,-176.506,7.120,148.312
C01389=1211.462,301.081,-68.004,-176.504,7.122,148.312
C01390=1211.457,301.329,-68.034,-176.502,7.125,148.312
C01391=1211.453,301.577,-68.064,-176.499,7.127,148.312
C01392=1211.449,301.826,-68.093,-176.497,7.130,148.312
C01393=1211.445,302.073,-68.123,-176.495,7.132,148.312
C01394=1211.441,302.322,-68.153,-176.492,7.135,148.312
C01395=1211.436,302.570,-68.182,-176.490,7.137,148.312
C01396=1211.432,302.818,-68.212,-176.487,7.140,148.312
C01397=1211.427,303.067,-68.242,-176.485,7.143,148.312
C01398=1211.423,303.315,-68.271,-176.482,7.146,148.312
C01399=1211.419,303.563,-68.301,-176.480,7.149,148.312
C01400=1211.414,303.811,-68.331,-176.478,7.151,148.312
C01401=1211.410,304.060,-68.361,-176.475,7.154,148.312
C01402=1211.405,304.307,-68.390,-176.473,7.156,148.312
C01403=1211.402,304.555,-68.420,-176.470,7.159,148.312
C01404=1211.397,304.804,-68.450,-176.468,7.161,148.312
C01405=1211.393,305.052,-68.480,-176.465,7.164,148.312
C01406=1211.389,305.300,-68.510,-176.463,7.167,148.312
C01407=1211.384,305.549,-68.540,-176.460,7.170,148.312
C01408=1211.380,305.797,-68.570,-176.458,7.172,148.312
C01409=1211.376,306.044,-68.600,-176.456,7.175,148.312
C01410=1211.371,306.293,-68.630,-176.454,7.177,148.311
C01411=1211.367,306.541,-68.659,-176.451,7.180,148.311
C01412=1211.363,306.789,-68.689,-176.449,7.182,148.311
C01413=1211.358,307.037,-68.719,-176.446,7.185,148.311
C01414=1211.354,307.285,-68.750,-176.444,7.188,148.311
C01415=1211.350,307.533,-68.779,-176.441,7.191,148.311
C01416=1211.345,307.782,-68.809,-176.439,7.193,148.311
C01417=1211.341,308.030,-68.839,-176.436,7.196,148.311
C01418=1211.337,308.278,-68.869,-176.434,7.198,148.311
C01419=1211.333,308.526,-68.900,-176.432,7.201,148.311
C01420=1211.328,308.774,-68.929,-176.430,7.204,148.311
C01421=1211.324,309.022,-68.960,-176.427,7.207,148.311
C01422=1211.320,309.270,-68.989,-176.425,7.209,148.311
C01423=1211.316,309.519,-69.020,-176.423,7.212,148.311
C01424=1211.311,309.767,-69.050,-176.420,7.215,148.311
C01425=1211.308,310.015,-69.080,-176.418,7.217,148.311
C01426=1211.303,310.264,-69.110,-176.415,7.220,148.311
C01427=1211.299,310.511,-69.140,-176.413,7.222,148.311
C01428=1211.294,310.759,-69.171,-176.410,7.225,148.311
C01429=1211.290,311.007,-69.200,-176.409,7.228,148.311
C01430=1211.285,311.255,-69.231,-176.406,7.231,148.311
C01431=1211.281,311.504,-69.261,-176.404,7.233,148.311
C01432=1211.277,311.752,-69.292,-176.401,7.236,148.311
C01433=1211.273,312.000,-69.322,-176.399,7.238,148.311
C01434=1211.268,312.248,-69.352,-176.396,7.241,148.311
C01435=1211.265,312.496,-69.382,-176.394,7.244,148.311
C01436=1211.260,312.744,-69.413,-176.392,7.247,148.311
C01437=1211.256,312.992,-69.442,-176.390,7.249,148.311
C01438=1211.252,313.241,-69.473,-176.387,7.252,148.311
C01439=1211.248,313.489,-69.504,-176.385,7.255,148.311
C01440=1211.243,313.737,-69.534,-176.382,7.258,148.311
C01441=1211.239,313.985,-69.564,-176.380,7.261,148.311
C01442=1211.234,314.233,-69.595,-176.378,7.263,148.311
C01443=1211.231,314.480,-69.625,-176.375,7.266,148.311
C01444=1211.226,314.758,-69.659,-176.373,7.269,148.311
C01445=1211.221,315.033,-69.693,-176.370,7.272,148.311
C01446=1211.216,315.310,-69.727,-176.367,7.275,148.311
C01447=1211.211,315.586,-69.761,-176.365,7.277,148.311
C01448=1211.208,315.833,-69.791,-176.363,7.280,148.311
C01449=1211.203,316.081,-69.822,-176.360,7.284,148.312
C01450=1211.198,316.329,-69.853,-176.358,7.286,148.311
C01451=1211.195,316.578,-69.882,-176.356,7.289,148.311
C01452=1211.190,316.826,-69.913,-176.354,7.291,148.311
C01453=1211.186,317.074,-69.944,-176.351,7.295,148.312
C01454=1211.182,317.322,-69.974,-176.349,7.297,148.312
C01455=1211.178,317.570,-70.005,-176.347,7.300,148.312
C01456=1211.173,317.818,-70.036,-176.344,7.302,148.312
C01457=1211.169,318.066,-70.066,-176.342,7.305,148.312
C01458=1211.165,318.314,-70.097,-176.340,7.308,148.312
C01459=1211.161,318.563,-70.128,-176.337,7.311,148.312
C01460=1211.157,318.810,-70.158,-176.335,7.314,148.312
C01461=1211.152,319.058,-70.189,-176.333,7.316,148.312
C01462=1211.148,319.307,-70.220,-176.330,7.319,148.312
C01463=1211.144,319.554,-70.250,-176.328,7.321,148.312
C01464=1211.140,319.802,-70.281,-176.326,7.325,148.312
C01465=1211.135,320.050,-70.312,-176.324,7.327,148.312
C01466=1211.131,320.299,-70.343,-176.321,7.330,148.312
C01467=1211.127,320.547,-70.373,-176.319,7.333,148.312
C01468=1211.122,320.795,-70.404,-176.317,7.336,148.312
C01469=1211.118,321.043,-70.435,-176.314,7.339,148.312
C01470=1211.114,321.291,-70.466,-176.312,7.341,148.312
C01471=1211.109,321.539,-70.496,-176.310,7.344,148.312
C01472=1211.106,321.788,-70.527,-176.308,7.346,148.312
C01473=1211.101,322.036,-70.558,-176.305,7.349,148.312
C01474=1211.097,322.283,-70.589,-176.304,7.352,148.312
C01475=1211.093,322.532,-70.620,-176.301,7.355,148.312
C01476=1211.088,322.780,-70.651,-176.298,7.358,148.312
C01477=1211.084,323.027,-70.681,-176.297,7.361,148.313
C01478=1211.080,323.276,-70.712,-176.294,7.364,148.313
C01479=1211.076,323.524,-70.743,-176.292,7.366,148.313
C01480=1211.072,323.771,-70.775,-176.290,7.369,148.313
C01481=1211.068,324.020,-70.806,-176.287,7.371,148.313
C01482=1211.063,324.268,-70.837,-176.285,7.375,148.313
C01483=1211.059,324.516,-70.868,-176.283,7.377,148.313
C01484=1211.055,324.763,-70.899,-176.281,7.380,148.313
C01485=1211.051,325.011,-70.929,-176.278,7.383,148.313
C01486=1211.047,325.260,-70.960,-176.276,7.385,148.313
C01487=1211.042,325.507,-70.992,-176.274,7.389,148.313
C01488=1211.038,325.756,-71.023,-176.272,7.391,148.313
C01489=1211.034,326.004,-71.054,-176.270,7.394,148.313
C01490=1211.029,326.252,-71.085,-176.267,7.397,148.313
C01491=1211.025,326.500,-71.116,-176.265,7.400,148.314
C01492=1211.021,326.748,-71.147,-176.263,7.402,148.314
C01493=1211.017,326.996,-71.179,-176.260,7.405,148.314
C01494=1211.013,327.244,-71.210,-176.258,7.409,148.314
C01495=1211.009,327.493,-71.241,-176.256,7.411,148.314
C01496=1211.004,327.740,-71.272,-176.254,7.414,148.314
C01497=1211.000,327.988,-71.303,-176.252,7.416,148.314
C01498=1210.996,328.236,-71.335,-176.250,7.420,148.314
C01499=1210.991,328.484,-71.366,-176.247,7.422,148.314
C01500=1210.987,328.733,-71.397,-176.245,7.425,148.314
C01501=1210.983,328.980,-71.428,-176.243,7.428,148.314
C01502=1210.979,329.229,-71.460,-176.241,7.431,148.314
C01503=1210.975,329.476,-71.491,-176.238,7.434,148.315
C01504=1210.971,329.725,-71.522,-176.237,7.436,148.315
C01505=1210.966,329.972,-71.554,-176.234,7.439,148.315
C01506=1210.962,330.221,-71.585,-176.232,7.442,148.315
C01507=1210.958,330.468,-71.616,-176.230,7.445,148.315
C01508=1210.954,330.717,-71.647,-176.228,7.447,148.315
C01509=1210.950,330.964,-71.679,-176.225,7.450,148.315
C01510=1210.946,331.212,-71.711,-176.223,7.454,148.315
C01511=1210.941,331.460,-71.741,-176.221,7.456,148.315
C01512=1210.938,331.708,-71.773,-176.219,7.459,148.315
C01513=1210.933,331.956,-71.804,-176.217,7.462,148.316
C01514=1210.929,332.204,-71.837,-176.214,7.465,148.316
C01515=1210.924,332.452,-71.867,-176.213,7.467,148.316
C01516=1210.920,332.700,-71.899,-176.211,7.471,148.316
C01517=1210.916,332.948,-71.931,-176.208,7.473,148.316
C01518=1210.912,333.196,-71.962,-176.206,7.476,148.316
C01519=1210.908,333.444,-71.993,-176.204,7.479,148.316
C01520=1210.904,333.692,-72.025,-176.202,7.482,148.316
C01521=1210.899,333.940,-72.056,-176.200,7.485,148.317
C01522=1210.895,334.188,-72.088,-176.198,7.487,148.317
C01523=1210.891,334.435,-72.120,-176.195,7.491,148.317
C01524=1210.887,334.683,-72.152,-176.193,7.493,148.317
C01525=1210.883,334.932,-72.183,-176.191,7.496,148.317
C01526=1210.878,335.180,-72.215,-176.189,7.499,148.317
C01527=1210.874,335.428,-72.247,-176.187,7.502,148.317
C01528=1210.870,335.675,-72.278,-176.185,7.505,148.317
C01529=1210.866,335.924,-72.309,-176.183,7.508,148.318
C01530=1210.862,336.172,-72.341,-176.180,7.511,148.318
C01531=1210.857,336.419,-72.373,-176.179,7.513,148.318
C01532=1210.853,336.667,-72.405,-176.176,7.517,148.318
C01533=1210.849,336.915,-72.436,-176.175,7.519,148.318
C01534=1210.845,337.163,-72.469,-176.172,7.522,148.318
C01535=1210.841,337.412,-72.500,-176.170,7.525,148.318
C01536=1210.836,337.659,-72.532,-176.168,7.528,148.318
C01537=1210.833,337.907,-72.563,-176.166,7.531,148.319
C01538=1210.828,338.155,-72.595,-176.164,7.534,148.319
C01539=1210.824,338.403,-72.627,-176.162,7.537,148.319
C01540=1210.820,338.651,-72.659,-176.160,7.540,148.319
C01541=1210.815,338.898,-72.691,-176.157,7.543,148.319
C01542=1210.811,339.146,-72.723,-176.156,7.545,148.319
C01543=1210.808,339.395,-72.755,-176.154,7.548,148.319
C01544=1210.803,339.642,-72.787,-176.152,7.551,148.320
C01545=1210.799,339.890,-72.819,-176.150,7.554,148.320
C01546=1210.795,340.138,-72.851,-176.148,7.556,148.320
C01547=1210.790,340.386,-72.883,-176.145,7.560,148.320
C01548=1210.786,340.665,-72.918,-176.143,7.563,148.320
C01549=1210.781,340.943,-72.954,-176.141,7.567,148.321
C01550=1210.777,341.220,-72.990,-176.138,7.570,148.321
C01551=1210.771,341.499,-73.025,-176.136,7.573,148.321
C01552=1210.768,341.746,-73.058,-176.134,7.575,148.321
C01553=1210.764,341.994,-73.090,-176.132,7.579,148.321
C01554=1210.759,342.242,-73.122,-176.131,7.581,148.321
C01555=1210.755,342.490,-73.154,-176.128,7.585,148.322
C01556=1210.751,342.738,-73.186,-176.126,7.588,148.322
C01557=1210.746,342.986,-73.218,-176.124,7.590,148.322
C01558=1210.742,343.234,-73.250,-176.122,7.594,148.322
C01559=1210.738,343.482,-73.282,-176.120,7.596,148.322
C01560=1210.734,343.730,-73.314,-176.118,7.599,148.322
C01561=1210.729,343.977,-73.347,-176.116,7.602,148.323
C01562=1210.726,344.225,-73.379,-176.114,7.605,148.323
C01563=1210.722,344.473,-73.411,-176.112,7.608,148.323
C01564=1210.718,344.722,-73.443,-176.110,7.611,148.323
C01565=1210.713,344.969,-73.475,-176.109,7.614,148.323
C01566=1210.709,345.217,-73.508,-176.106,7.617,148.324
C01567=1210.705,345.465,-73.540,-176.105,7.620,148.324
C01568=1210.700,345.712,-73.572,-176.103,7.623,148.324
C01569=1210.696,345.961,-73.604,-176.101,7.625,148.324
C01570=1210.692,346.209,-73.636,-176.098,7.628,148.324
C01571=1210.688,346.456,-73.669,-176.097,7.631,148.324
C01572=1210.684,346.705,-73.701,-176.094,7.634,148.325
C01573=1210.679,346.952,-73.733,-176.092,7.638,148.325
C01574=1210.676,347.200,-73.766,-176.090,7.640,148.325
C01575=1210.671,347.448,-73.798,-176.088,7.644,148.325
C01576=1210.667,347.696,-73.831,-176.087,7.646,148.325
C01577=1210.663,347.943,-73.863,-176.085,7.650,148.326
C01578=1210.659,348.191,-73.895,-176.083,7.652,148.326
C01579=1210.655,348.439,-73.927,-176.081,7.656,148.326
C01580=1210.651,348.687,-73.960,-176.079,7.658,148.326
C01581=1210.646,348.935,-73.993,-176.077,7.661,148.327
C01582=1210.642,349.182,-74.025,-176.076,7.664,148.327
C01583=1210.638,349.431,-74.057,-176.073,7.667,148.327
C01584=1210.634,349.679,-74.089,-176.072,7.670,148.327
C01585=1210.630,349.926,-74.122,-176.069,7.673,148.327
C01586=1210.626,350.175,-74.155,-176.068,7.676,148.328
C01587=1210.622,350.422,-74.187,-176.066,7.679,148.328
C01588=1210.617,350.670,-74.219,-176.064,7.682,148.328
C01589=1210.613,350.917,-74.253,-176.062,7.685,148.328
C01590=1210.609,351.165,-74.284,-176.061,7.688,148.329
C01591=1210.605,351.413,-74.318,-176.058,7.691,148.329
C01592=1210.601,351.662,-74.350,-176.057,7.694,148.329
C01593=1210.597,351.909,-74.383,-176.054,7.697,148.329
C01594=1210.593,352.157,-74.415,-176.053,7.699,148.329
C01595=1210.588,352.404,-74.448,-176.051,7.703,148.330
C01596=1210.584,352.653,-74.480,-176.049,7.706,148.330
C01597=1210.580,352.900,-74.513,-176.047,7.709,148.330
C01598=1210.576,353.148,-74.545,-176.046,7.711,148.331
C01599=1210.572,353.396,-74.578,-176.043,7.715,148.331
C01600=1210.568,353.644,-74.611,-176.042,7.717,148.331
C01601=1210.564,353.892,-74.643,-176.040,7.721,148.331
C01602=1210.560,354.140,-74.676,-176.038,7.723,148.332
C01603=1210.555,354.388,-74.709,-176.036,7.727,148.332
C01604=1210.551,354.635,-74.742,-176.034,7.729,148.332
C01605=1210.547,354.883,-74.774,-176.033,7.733,148.332
C01606=1210.543,355.131,-74.807,-176.031,7.735,148.333
C01607=1210.539,355.379,-74.840,-176.029,7.738,148.333
C01608=1210.534,355.626,-74.873,-176.027,7.741,148.333
C01609=1210.530,355.875,-74.905,-176.026,7.744,148.333
C01610=1210.527,356.122,-74.938,-176.024,7.747,148.334
C01611=1210.522,356.370,-74.971,-176.022,7.750,148.334
C01612=1210.518,356.618,-75.004,-176.020,7.754,148.334
C01613=1210.514,356.866,-75.037,-176.019,7.756,148.334
C01614=1210.510,357.114,-75.070,-176.017,7.760,148.335
C01615=1210.506,357.361,-75.103,-176.015,7.762,148.335
C01616=1210.502,357.609,-75.136,-176.013,7.766,148.335
C01617=1210.498,357.857,-75.168,-176.011,7.768,148.335
C01618=1210.494,358.105,-75.201,-176.010,7.772,148.336
C01619=1210.489,358.353,-75.234,-176.008,7.774,148.336
C01620=1210.485,358.600,-75.268,-176.007,7.777,148.336
C01621=1210.481,358.847,-75.300,-176.005,7.781,148.337
C01622=1210.476,359.095,-75.334,-176.003,7.783,148.337
C01623=1210.472,359.343,-75.366,-176.001,7.787,148.337
C01624=1210.469,359.591,-75.399,-176.000,7.789,148.337
C01625=1210.464,359.839,-75.432,-175.998,7.793,148.338
C01626=1210.460,360.086,-75.465,-175.996,7.795,148.338
C01627=1210.456,360.334,-75.498,-175.994,7.799,148.339
C01628=1210.452,360.582,-75.531,-175.993,7.802,148.339
C01629=1210.448,360.829,-75.564,-175.991,7.804,148.339
C01630=1210.444,361.077,-75.597,-175.989,7.808,148.339
C01631=1210.440,361.326,-75.631,-175.988,7.810,148.340
C01632=1210.436,361.573,-75.664,-175.986,7.814,148.340
C01633=1210.432,361.821,-75.697,-175.985,7.817,148.340
C01634=1210.428,362.069,-75.730,-175.983,7.819,148.341
C01635=1210.423,362.317,-75.763,-175.981,7.823,148.341
C01636=1210.419,362.565,-75.796,-175.980,7.825,148.341
C01637=1210.415,362.813,-75.829,-175.978,7.829,148.342
C01638=1210.411,363.060,-75.862,-175.976,7.832,148.342
C01639=1210.407,363.308,-75.896,-175.975,7.834,148.342
C01640=1210.403,363.555,-75.929,-175.973,7.838,148.343
C01641=1210.399,363.803,-75.963,-175.972,7.840,148.343
C01642=1210.395,364.051,-75.996,-175.971,7.843,148.343
C01643=1210.391,364.298,-76.029,-175.968,7.847,148.343
C01644=1210.386,364.546,-76.062,-175.967,7.849,148.344
C01645=1210.382,364.794,-76.095,-175.965,7.853,148.344
C01646=1210.378,365.042,-76.128,-175.964,7.856,148.344
C01647=1210.374,365.289,-76.161,-175.963,7.858,148.345
C01648=1210.370,365.538,-76.195,-175.961,7.862,148.345
C01649=1210.366,365.785,-76.228,-175.959,7.865,148.345
C01650=1210.362,366.033,-76.261,-175.958,7.867,148.346
C01651=1210.358,366.280,-76.295,-175.957,7.870,148.346
C01652=1210.353,366.561,-76.333,-175.955,7.874,148.347
C01653=1210.349,366.841,-76.370,-175.953,7.877,148.347
C01654=1210.344,367.121,-76.408,-175.951,7.881,148.347
C01655=1210.339,367.402,-76.446,-175.950,7.884,148.348
C01656=1210.335,367.649,-76.480,-175.948,7.887,148.348
C01657=1210.331,367.897,-76.513,-175.947,7.890,148.349
C01658=1210.327,368.145,-76.546,-175.945,7.893,148.349
C01659=1210.323,368.392,-76.579,-175.943,7.896,148.349
C01660=1210.319,368.640,-76.614,-175.942,7.899,148.350
C01661=1210.315,368.888,-76.647,-175.941,7.902,148.350
C01662=1210.311,369.136,-76.680,-175.940,7.905,148.350
C01663=1210.306,369.384,-76.713,-175.938,7.908,148.351
C01664=1210.303,369.631,-76.747,-175.936,7.911,148.351
C01665=1210.298,369.878,-76.780,-175.935,7.914,148.351
C01666=1210.294,370.126,-76.814,-175.934,7.917,148.352
C01667=1210.290,370.375,-76.848,-175.932,7.920,148.352
C01668=1210.286,370.622,-76.882,-175.931,7.923,148.353
C01669=1210.282,370.870,-76.915,-175.930,7.926,148.353
C01670=1210.278,371.117,-76.948,-175.929,7.929,148.353
C01671=1210.273,371.365,-76.982,-175.928,7.931,148.354
C01672=1210.269,371.613,-77.016,-175.926,7.935,148.354
C01673=1210.266,371.860,-77.050,-175.925,7.938,148.355
C01674=1210.262,372.108,-77.083,-175.923,7.941,148.355
C01675=1210.257,372.356,-77.117,-175.922,7.944,148.355
C01676=1210.253,372.603,-77.151,-175.921,7.946,148.356
C01677=1210.249,372.851,-77.184,-175.920,7.949,148.356
C01678=1210.246,373.099,-77.217,-175.918,7.953,148.357
C01679=1210.241,373.347,-77.252,-175.917,7.956,148.357
C01680=1210.237,373.595,-77.285,-175.916,7.958,148.357
C01681=1210.233,373.842,-77.319,-175.914,7.961,148.358
C01682=1210.229,374.089,-77.352,-175.913,7.964,148.358
C01683=1210.225,374.338,-77.387,-175.912,7.967,148.359
C01684=1210.221,374.585,-77.420,-175.911,7.970,148.359
C01685=1210.217,374.832,-77.454,-175.910,7.972,148.359
C01686=1210.212,375.080,-77.487,-175.908,7.976,148.360
C01687=1210.208,375.328,-77.521,-175.907,7.979,148.360
C01688=1210.205,375.576,-77.555,-175.905,7.982,148.361
C01689=1210.201,375.823,-77.589,-175.904,7.985,148.361
C01690=1210.196,376.071,-77.622,-175.903,7.987,148.361
C01691=1210.192,376.318,-77.656,-175.902,7.990,148.362
C01692=1210.189,376.567,-77.690,-175.901,7.993,148.362
C01693=1210.184,376.814,-77.724,-175.900,7.996,148.363
C01694=1210.180,377.062,-77.758,-175.899,7.999,148.363
C01695=1210.175,377.309,-77.792,-175.898,8.002,148.364
C01696=1210.172,377.558,-77.825,-175.896,8.005,148.364
C01697=1210.168,377.805,-77.859,-175.895,8.007,148.364
C01698=1210.163,378.052,-77.894,-175.894,8.010,148.365
C01699=1210.159,378.300,-77.927,-175.893,8.013,148.365
C01700=1210.156,378.548,-77.961,-175.892,8.016,148.366
C01701=1210.151,378.796,-77.995,-175.891,8.019,148.366
C01702=1210.147,379.043,-78.029,-175.890,8.022,148.367
C01703=1210.143,379.290,-78.063,-175.889,8.025,148.367
C01704=1210.139,379.539,-78.097,-175.888,8.028,148.368
C01705=1210.135,379.786,-78.131,-175.886,8.030,148.368
C01706=1210.131,380.033,-78.165,-175.886,8.034,148.369
C01707=1210.127,380.282,-78.199,-175.884,8.036,148.369
C01708=1210.123,380.529,-78.233,-175.883,8.039,148.369
C01709=1210.119,380.776,-78.267,-175.882,8.042,148.370
C01710=1210.114,381.024,-78.301,-175.881,8.045,148.370
C01711=1210.111,381.272,-78.335,-175.880,8.048,148.371
C01712=1210.107,381.519,-78.369,-175.879,8.051,148.371
C01713=1210.102,381.767,-78.403,-175.878,8.054,148.372
C01714=1210.099,382.015,-78.437,-175.877,8.056,148.372
C01715=1210.094,382.262,-78.471,-175.876,8.059,148.372
C01716=1210.090,382.510,-78.505,-175.876,8.062,148.373
C01717=1210.086,382.758,-78.539,-175.874,8.065,148.373
C01718=1210.082,383.005,-78.573,-175.873,8.067,148.374
C01719=1210.078,383.253,-78.608,-175.872,8.070,148.374
C01720=1210.074,383.501,-78.642,-175.871,8.073,148.375
C01721=1210.070,383.748,-78.676,-175.870,8.076,148.375
C01722=1210.066,383.996,-78.710,-175.870,8.078,148.376
C01723=1210.062,384.244,-78.744,-175.869,8.081,148.376
C01724=1210.058,384.491,-78.778,-175.868,8.084,148.377
C01725=1210.053,384.738,-78.813,-175.867,8.087,148.377
C01726=1210.050,384.986,-78.847,-175.866,8.090,148.378
C01727=1210.045,385.234,-78.881,-175.865,8.092,148.378
C01728=1210.041,385.481,-78.915,-175.864,8.095,148.378
C01729=1210.037,385.729,-78.949,-175.863,8.098,148.379
C01730=1210.034,385.977,-78.983,-175.862,8.101,148.379
C01731=1210.029,386.224,-79.018,-175.862,8.103,148.380
C01732=1210.026,386.472,-79.052,-175.861,8.106,148.380
C01733=1210.021,386.719,-79.086,-175.860,8.109,148.381
C01734=1210.016,386.967,-79.120,-175.859,8.112,148.381
C01735=1210.013,387.215,-79.154,-175.858,8.114,148.382
C01736=1210.009,387.463,-79.189,-175.857,8.117,148.382
C01737=1210.005,387.710,-79.223,-175.857,8.120,148.383
C01738=1210.001,387.958,-79.258,-175.855,8.123,148.383
C01739=1209.997,388.205,-79.291,-175.855,8.125,148.384
C01740=1209.993,388.453,-79.326,-175.854,8.128,148.384
C01741=1209.988,388.700,-79.361,-175.853,8.131,148.385
C01742=1209.985,388.947,-79.395,-175.852,8.133,148.385
C01743=1209.981,389.196,-79.429,-175.852,8.136,148.386
C01744=1209.977,389.443,-79.463,-175.851,8.139,148.386
C01745=1209.973,389.691,-79.498,-175.850,8.141,148.387
C01746=1209.968,389.938,-79.533,-175.849,8.144,148.387
C01747=1209.964,390.185,-79.567,-175.848,8.147,148.388
C01748=1209.960,390.433,-79.601,-175.848,8.149,148.388
C01749=1209.957,390.681,-79.635,-175.847,8.152,148.389
C01750=1209.953,390.929,-79.670,-175.847,8.155,148.389
C01751=1209.948,391.176,-79.705,-175.846,8.157,148.389
C01752=1209.945,391.424,-79.739,-175.845,8.160,148.390
C01753=1209.940,391.671,-79.773,-175.844,8.162,148.390
C01754=1209.936,391.919,-79.808,-175.843,8.166,148.391
C01755=1209.932,392.167,-79.842,-175.843,8.168,148.392
C01756=1209.927,392.449,-79.881,-175.842,8.171,148.392
C01757=1209.923,392.731,-79.920,-175.841,8.174,148.393
C01758=1209.918,393.014,-79.960,-175.840,8.177,148.393
C01759=1209.914,393.296,-79.999,-175.840,8.180,148.394
C01760=1209.910,393.544,-80.034,-175.839,8.182,148.394
C01761=1209.906,393.791,-80.068,-175.838,8.185,148.395
C01762=1209.902,394.039,-80.103,-175.838,8.187,148.395
C01763=1209.897,394.287,-80.137,-175.837,8.190,148.396
C01764=1209.893,394.534,-80.171,-175.837,8.192,148.396
C01765=1209.889,394.782,-80.206,-175.836,8.195,148.397
C01766=1209.885,395.029,-80.241,-175.835,8.197,148.397
C01767=1209.882,395.276,-80.275,-175.834,8.201,148.398
C01768=1209.877,395.524,-80.310,-175.834,8.203,148.398
C01769=1209.873,395.772,-80.344,-175.833,8.206,148.399
C01770=1209.869,396.019,-80.379,-175.833,8.208,148.399
C01771=1209.866,396.267,-80.413,-175.832,8.211,148.400
C01772=1209.861,396.515,-80.448,-175.831,8.213,148.400
C01773=1209.857,396.762,-80.483,-175.831,8.216,148.401
C01774=1209.853,397.010,-80.518,-175.830,8.218,148.401
C01775=1209.849,397.257,-80.552,-175.830,8.220,148.402
C01776=1209.845,397.505,-80.586,-175.829,8.223,148.402
C01777=1209.840,397.752,-80.621,-175.828,8.225,148.402
C01778=1209.837,398.000,-80.656,-175.828,8.228,148.403
C01779=1209.833,398.247,-80.690,-175.827,8.231,148.404
C01780=1209.829,398.495,-80.725,-175.827,8.233,148.404
C01781=1209.824,398.742,-80.760,-175.826,8.236,148.405
C01782=1209.820,398.990,-80.794,-175.826,8.238,148.405
C01783=1209.817,399.237,-80.829,-175.825,8.240,148.405
C01784=1209.813,399.485,-80.864,-175.824,8.243,148.406
C01785=1209.808,399.732,-80.898,-175.824,8.245,148.407
C01786=1209.804,399.981,-80.933,-175.824,8.247,148.407
C01787=1209.800,400.227,-80.968,-175.823,8.251,148.407
C01788=1209.797,400.475,-81.003,-175.823,8.253,148.408
C01789=1209.792,400.723,-81.037,-175.822,8.255,148.408
C01790=1209.788,400.971,-81.072,-175.821,8.258,148.409
C01791=1209.784,401.218,-81.107,-175.821,8.260,148.409
C01792=1209.780,401.466,-81.142,-175.820,8.262,148.410
C01793=1209.776,401.713,-81.176,-175.820,8.264,148.410
C01794=1209.772,401.961,-81.211,-175.819,8.268,148.411
C01795=1209.768,402.208,-81.246,-175.819,8.269,148.411
C01796=1209.764,402.456,-81.281,-175.818,8.272,148.412
C01797=1209.760,402.703,-81.315,-175.818,8.275,148.412
C01798=1209.757,402.950,-81.350,-175.817,8.277,148.413
C01799=1209.753,403.199,-81.385,-175.817,8.279,148.413
C01800=1209.748,403.446,-81.419,-175.817,8.281,148.414
C01801=1209.744,403.693,-81.455,-175.816,8.284,148.414
C01802=1209.740,403.941,-81.489,-175.815,8.286,148.415
C01803=1209.736,404.189,-81.524,-175.815,8.289,148.415
C01804=1209.732,404.436,-81.559,-175.815,8.291,148.416
C01805=1209.728,404.684,-81.594,-175.814,8.293,148.416
C01806=1209.724,404.931,-81.628,-175.813,8.296,148.417
C01807=1209.720,405.179,-81.664,-175.813,8.298,148.417
C01808=1209.716,405.426,-81.698,-175.812,8.300,148.418
C01809=1209.712,405.673,-81.734,-175.812,8.303,148.418
C01810=1209.707,405.921,-81.768,-175.812,8.305,148.419
C01811=1209.703,406.169,-81.803,-175.811,8.307,148.419
C01812=1209.700,406.416,-81.838,-175.811,8.310,148.420
C01813=1209.696,406.664,-81.872,-175.810,8.312,148.420
C01814=1209.692,406.911,-81.908,-175.810,8.314,148.420
C01815=1209.688,407.159,-81.942,-175.810,8.316,148.421
C01816=1209.684,407.407,-81.977,-175.809,8.319,148.422
C01817=1209.679,407.653,-82.012,-175.809,8.321,148.422
C01818=1209.675,407.902,-82.047,-175.808,8.323,148.422
